// TIA Portal project "Boiler_DE_10_14GM" (V14)
// Паровой котел ДЕ-10-14ГМ

(* hardware
DEVICE "ET 200SP station_1"  ET 200SP-Station
   slot 0: "Rack_0"  Rack  6ES5 710-8MAx1
   slot 1: "PLC_1"  CPU 1510SP-1 PN  6ES7 510-1DJ01-0AB0  V2.1
   slot 2: "AI 8xI 2-,4-wire BA_1"  AI 8xI 2-,4-wire BA  6ES7 134-6GF00-0AA1  V1.0
      slot 1: "AI 8xI 2-,4-wire BA_1"  AI 8xI 2-,4-wire BA
   slot 3: "AI 8xI 2-,4-wire BA_2"  AI 8xI 2-,4-wire BA  6ES7 134-6GF00-0AA1  V1.0
      slot 1: "AI 8xI 2-,4-wire BA_2"  AI 8xI 2-,4-wire BA
   slot 4: "AI 8xI 2-,4-wire BA_3"  AI 8xI 2-,4-wire BA  6ES7 134-6GF00-0AA1  V1.0
      slot 1: "AI 8xI 2-,4-wire BA_3"  AI 8xI 2-,4-wire BA
   slot 5: "AI 8xI 2-,4-wire BA_4"  AI 8xI 2-,4-wire BA  6ES7 134-6GF00-0AA1  V1.0
      slot 1: "AI 8xI 2-,4-wire BA_4"  AI 8xI 2-,4-wire BA
   slot 6: "DI 16x24VDC ST_1"  DI 16x24VDC ST  6ES7 131-6BH00-0BA0  V1.1
      slot 1: "DI 16x24VDC ST_1"  DI 16x24VDC ST
   slot 7: "DI 16x24VDC ST_2"  DI 16x24VDC ST  6ES7 131-6BH00-0BA0  V1.1
      slot 1: "DI 16x24VDC ST_2"  DI 16x24VDC ST
   slot 8: "DI 16x24VDC ST_3"  DI 16x24VDC ST  6ES7 131-6BH00-0BA0  V1.1
      slot 1: "DI 16x24VDC ST_3"  DI 16x24VDC ST
   slot 9: "DI 16x24VDC ST_4"  DI 16x24VDC ST  6ES7 131-6BH00-0BA0  V1.1
      slot 1: "DI 16x24VDC ST_4"  DI 16x24VDC ST
   slot 10: "DI 16x24VDC ST_5"  DI 16x24VDC ST  6ES7 131-6BH00-0BA0  V1.1
      slot 1: "DI 16x24VDC ST_5"  DI 16x24VDC ST
   slot 11: "DI 16x24VDC ST_6"  DI 16x24VDC ST  6ES7 131-6BH00-0BA0  V1.1
      slot 1: "DI 16x24VDC ST_6"  DI 16x24VDC ST
   slot 12: "DQ 16x24VDC/0.5A ST_1"  DQ 16x24VDC/0.5A ST  6ES7 132-6BH00-0BA0  V1.1
      slot 1: "DQ 16x24VDC/0.5A ST_1"  DQ 16x24VDC/0.5A ST
   slot 13: "DQ 16x24VDC/0.5A ST_2"  DQ 16x24VDC/0.5A ST  6ES7 132-6BH00-0BA0  V1.1
      slot 1: "DQ 16x24VDC/0.5A ST_2"  DQ 16x24VDC/0.5A ST
   slot 14: "DQ 16x24VDC/0.5A ST_3"  DQ 16x24VDC/0.5A ST  6ES7 132-6BH00-0BA0  V1.1
      slot 1: "DQ 16x24VDC/0.5A ST_3"  DQ 16x24VDC/0.5A ST
   slot 15: "AQ 4xU/I ST_1"  AQ 4xU/I ST  6ES7 135-6HD00-0BA1  V1.1
      slot 1: "AQ 4xU/I ST_1"  AQ 4xU/I ST
   slot 16: "Server module_1"  Server module  6ES7 193-6PA00-0AA0  V1.1
      slot 1: "Server module_1"  Server module
   slot 127: "BA 2xRJ45"  BA 2xRJ45  6ES7 193-6AR00-0AA0  V0.0
      slot 32769: "Port_1"  6ES7 193-6AR00-0AA0
      slot 32770: "Port_2"  6ES7 193-6AR00-0AA0
*)

// ===== PLC "PLC_1"  CPU 1510SP-1 PN =====

VAR_GLOBAL   // PLC tag table "Default tag table"
   "Module01Chanel1_DI" AT %I0.0 : Bool;
   "Module01Chanel2_DI" AT %I0.1 : Bool;
   "Module01Chanel3_DI" AT %I0.2 : Bool;
   "Module01Chanel4_DI" AT %I0.3 : Bool;
   "Module01Chanel5_DI" AT %I0.4 : Bool;
   "Module01Chanel6_DI" AT %I0.5 : Bool;
   "Module01Chanel7_DI" AT %I0.6 : Bool;
   "Module01Chanel8_DI" AT %I0.7 : Bool;
   "Module01Chanel9_DI" AT %I1.0 : Bool;
   "Module01Chanel10_DI" AT %I1.1 : Bool;
   "Module01Chanel11_DI" AT %I1.2 : Bool;
   "Module01Chanel12_DI" AT %I1.3 : Bool;
   "Module01Chanel13_DI" AT %I1.4 : Bool;
   "Module01Chanel14_DI" AT %I1.5 : Bool;
   "Module01Chanel15_DI" AT %I1.6 : Bool;
   "Module01Chanel16_DI" AT %I1.7 : Bool;
   "Module01Chanel1_DO" AT %Q0.0 : Bool;
   "Module01Chanel2_DO" AT %Q0.1 : Bool;
   "Module01Chanel3_DO" AT %Q0.2 : Bool;
   "Module01Chanel4_DO" AT %Q0.3 : Bool;
   "Module01Chanel5_DO" AT %Q0.4 : Bool;
   "Module01Chanel6_DO" AT %Q0.5 : Bool;
   "Module01Chanel7_DO" AT %Q0.6 : Bool;
   "Module01Chanel8_DO" AT %Q0.7 : Bool;
   "Module01Chanel9_DO" AT %Q1.0 : Bool;
   "Module01Chanel10_DO" AT %Q1.1 : Bool;
   "Module01Chanel11_DO" AT %Q1.2 : Bool;
   "Module01Chanel12_DO" AT %Q1.3 : Bool;
   "Module01Chanel13_DO" AT %Q1.4 : Bool;
   "Module01Chanel14_DO" AT %Q1.5 : Bool;
   "Module01Chanel15_DO" AT %Q1.6 : Bool;
   "Module01Chanel16_DO" AT %Q1.7 : Bool;
   "Module01Chanel1_AI" AT %IW0 : Int;
   "Module01Chanel2_AI" AT %IW2 : Int;
   "Module01Chanel3_AI" AT %IW4 : Int;
   "Module01Chanel4_AI" AT %IW6 : Int;
   "Module01Chanel5_AI" AT %IW8 : Int;
   "Module01Chanel6_AI" AT %IW10 : Int;
   "Module01Chanel7_AI" AT %IW12 : Int;
   "Module01Chanel8_AI" AT %IW14 : Int;
   "Module01Chanel1_AO" AT %QW0 : Int;
   "Module01Chanel2_AO" AT %QW2 : Int;
   "Module01Chanel3_AO" AT %QW4 : Int;
   "Module01Chanel4_AO" AT %QW6 : Int;
   "Module02Chanel1_DI" AT %I16.0 : Bool;
   "Module02Chanel2_DI" AT %I16.1 : Bool;
   "Module02Chanel3_DI" AT %I16.2 : Bool;
   "Module02Chanel4_DI" AT %I16.3 : Bool;
   "Module02Chanel5_DI" AT %I16.4 : Bool;
   "Module02Chanel6_DI" AT %I16.5 : Bool;
   "Module02Chanel7_DI" AT %I16.6 : Bool;
   "Module02Chanel8_DI" AT %I16.7 : Bool;
   "Module02Chanel9_DI" AT %I17.0 : Bool;
   "Module02Chanel10_DI" AT %I17.1 : Bool;
   "Module02Chanel11_DI" AT %I17.2 : Bool;
   "Module02Chanel12_DI" AT %I17.3 : Bool;
   "Module02Chanel13_DI" AT %I17.4 : Bool;
   "Module02Chanel14_DI" AT %I17.5 : Bool;
   "Module02Chanel15_DI" AT %I17.6 : Bool;
   "Module02Chanel16_DI" AT %I17.7 : Bool;
   "Module02Chanel1_DO" AT %Q16.0 : Bool;
   "Module02Chanel2_DO" AT %Q16.1 : Bool;
   "Module02Chanel3_DO" AT %Q16.2 : Bool;
   "Module02Chanel4_DO" AT %Q16.3 : Bool;
   "Module02Chanel5_DO" AT %Q16.4 : Bool;
   "Module02Chanel6_DO" AT %Q16.5 : Bool;
   "Module02Chanel7_DO" AT %Q16.6 : Bool;
   "Module02Chanel8_DO" AT %Q16.7 : Bool;
   "Module02Chanel9_DO" AT %Q17.0 : Bool;
   "Module02Chanel10_DO" AT %Q17.1 : Bool;
   "Module02Chanel11_DO" AT %Q17.2 : Bool;
   "Module02Chanel12_DO" AT %Q17.3 : Bool;
   "Module02Chanel13_DO" AT %Q17.4 : Bool;
   "Module02Chanel14_DO" AT %Q17.5 : Bool;
   "Module02Chanel15_DO" AT %Q17.6 : Bool;
   "Module02Chanel16_DO" AT %Q17.7 : Bool;
   "Module02Chanel1_AI" AT %IW16 : Int;
   "Module02Chanel2_AI" AT %IW18 : Int;
   "Module02Chanel3_AI" AT %IW20 : Int;
   "Module02Chanel4_AI" AT %IW22 : Int;
   "Module02Chanel5_AI" AT %IW24 : Int;
   "Module02Chanel6_AI" AT %IW26 : Int;
   "Module02Chanel7_AI" AT %IW28 : Int;
   "Module02Chanel8_AI" AT %IW30 : Int;
   "Module02Chanel1_AO" AT %QW16 : Int;
   "Module02Chanel2_AO" AT %QW18 : Int;
   "Module02Chanel3_AO" AT %QW20 : Int;
   "Module02Chanel4_AO" AT %QW22 : Int;
   "Module03Chanel1_DI" AT %I32.0 : Bool;
   "Module03Chanel2_DI" AT %I32.1 : Bool;
   "Module03Chanel3_DI" AT %I32.2 : Bool;
   "Module03Chanel4_DI" AT %I32.3 : Bool;
   "Module03Chanel5_DI" AT %I32.4 : Bool;
   "Module03Chanel6_DI" AT %I32.5 : Bool;
   "Module03Chanel7_DI" AT %I32.6 : Bool;
   "Module03Chanel8_DI" AT %I32.7 : Bool;
   "Module03Chanel9_DI" AT %I33.0 : Bool;
   "Module03Chanel10_DI" AT %I33.1 : Bool;
   "Module03Chanel11_DI" AT %I33.2 : Bool;
   "Module03Chanel12_DI" AT %I33.3 : Bool;
   "Module03Chanel13_DI" AT %I33.4 : Bool;
   "Module03Chanel14_DI" AT %I33.5 : Bool;
   "Module03Chanel15_DI" AT %I33.6 : Bool;
   "Module03Chanel16_DI" AT %I33.7 : Bool;
   "Module03Chanel1_DO" AT %Q32.0 : Bool;
   "Module03Chanel2_DO" AT %Q32.1 : Bool;
   "Module03Chanel3_DO" AT %Q32.2 : Bool;
   "Module03Chanel4_DO" AT %Q32.3 : Bool;
   "Module03Chanel5_DO" AT %Q32.4 : Bool;
   "Module03Chanel6_DO" AT %Q32.5 : Bool;
   "Module03Chanel7_DO" AT %Q32.6 : Bool;
   "Module03Chanel8_DO" AT %Q32.7 : Bool;
   "Module03Chanel9_DO" AT %Q33.0 : Bool;
   "Module03Chanel10_DO" AT %Q33.1 : Bool;
   "Module03Chanel11_DO" AT %Q33.2 : Bool;
   "Module03Chanel12_DO" AT %Q33.3 : Bool;
   "Module03Chanel13_DO" AT %Q33.4 : Bool;
   "Module03Chanel14_DO" AT %Q33.5 : Bool;
   "Module03Chanel15_DO" AT %Q33.6 : Bool;
   "Module03Chanel16_DO" AT %Q33.7 : Bool;
   "Module03Chanel1_AI" AT %IW32 : Int;
   "Module03Chanel2_AI" AT %IW34 : Int;
   "Module03Chanel3_AI" AT %IW36 : Int;
   "Module03Chanel4_AI" AT %IW38 : Int;
   "Module03Chanel5_AI" AT %IW40 : Int;
   "Module03Chanel6_AI" AT %IW42 : Int;
   "Module03Chanel7_AI" AT %IW44 : Int;
   "Module03Chanel8_AI" AT %IW46 : Int;
   "Module03Chanel1_AO" AT %QW32 : Int;
   "Module03Chanel2_AO" AT %QW34 : Int;
   "Module03Chanel3_AO" AT %QW36 : Int;
   "Module03Chanel4_AO" AT %QW38 : Int;
   "Module04Chanel1_DI" AT %I48.0 : Bool;
   "Module04Chanel2_DI" AT %I48.1 : Bool;
   "Module04Chanel3_DI" AT %I48.2 : Bool;
   "Module04Chanel4_DI" AT %I48.3 : Bool;
   "Module04Chanel5_DI" AT %I48.4 : Bool;
   "Module04Chanel6_DI" AT %I48.5 : Bool;
   "Module04Chanel7_DI" AT %I48.6 : Bool;
   "Module04Chanel8_DI" AT %I48.7 : Bool;
   "Module04Chanel9_DI" AT %I49.0 : Bool;
   "Module04Chanel10_DI" AT %I49.1 : Bool;
   "Module04Chanel11_DI" AT %I49.2 : Bool;
   "Module04Chanel12_DI" AT %I49.3 : Bool;
   "Module04Chanel13_DI" AT %I49.4 : Bool;
   "Module04Chanel14_DI" AT %I49.5 : Bool;
   "Module04Chanel15_DI" AT %I49.6 : Bool;
   "Module04Chanel16_DI" AT %I49.7 : Bool;
   "Module04Chanel1_DO" AT %Q48.0 : Bool;
   "Module04Chanel2_DO" AT %Q48.1 : Bool;
   "Module04Chanel3_DO" AT %Q48.2 : Bool;
   "Module04Chanel4_DO" AT %Q48.3 : Bool;
   "Module04Chanel5_DO" AT %Q48.4 : Bool;
   "Module04Chanel6_DO" AT %Q48.5 : Bool;
   "Module04Chanel7_DO" AT %Q48.6 : Bool;
   "Module04Chanel8_DO" AT %Q48.7 : Bool;
   "Module04Chanel9_DO" AT %Q49.0 : Bool;
   "Module04Chanel10_DO" AT %Q49.1 : Bool;
   "Module04Chanel11_DO" AT %Q49.2 : Bool;
   "Module04Chanel12_DO" AT %Q49.3 : Bool;
   "Module04Chanel13_DO" AT %Q49.4 : Bool;
   "Module04Chanel14_DO" AT %Q49.5 : Bool;
   "Module04Chanel15_DO" AT %Q49.6 : Bool;
   "Module04Chanel16_DO" AT %Q49.7 : Bool;
   "Module04Chanel1_AI" AT %IW48 : Int;
   "Module04Chanel2_AI" AT %IW50 : Int;
   "Module04Chanel3_AI" AT %IW52 : Int;
   "Module04Chanel4_AI" AT %IW54 : Int;
   "Module04Chanel5_AI" AT %IW56 : Int;
   "Module04Chanel6_AI" AT %IW58 : Int;
   "Module04Chanel7_AI" AT %IW60 : Int;
   "Module04Chanel8_AI" AT %IW62 : Int;
   "Module04Chanel1_AO" AT %QW48 : Int;
   "Module04Chanel2_AO" AT %QW50 : Int;
   "Module04Chanel3_AO" AT %QW52 : Int;
   "Module04Chanel4_AO" AT %QW54 : Int;
   "Module05Chanel1_DI" AT %I64.0 : Bool;
   "Module05Chanel2_DI" AT %I64.1 : Bool;
   "Module05Chanel3_DI" AT %I64.2 : Bool;
   "Module05Chanel4_DI" AT %I64.3 : Bool;
   "Module05Chanel5_DI" AT %I64.4 : Bool;
   "Module05Chanel6_DI" AT %I64.5 : Bool;
   "Module05Chanel7_DI" AT %I64.6 : Bool;
   "Module05Chanel8_DI" AT %I64.7 : Bool;
   "Module05Chanel9_DI" AT %I65.0 : Bool;
   "Module05Chanel10_DI" AT %I65.1 : Bool;
   "Module05Chanel11_DI" AT %I65.2 : Bool;
   "Module05Chanel12_DI" AT %I65.3 : Bool;
   "Module05Chanel13_DI" AT %I65.4 : Bool;
   "Module05Chanel14_DI" AT %I65.5 : Bool;
   "Module05Chanel15_DI" AT %I65.6 : Bool;
   "Module05Chanel16_DI" AT %I65.7 : Bool;
   "Module05Chanel1_DO" AT %Q64.0 : Bool;
   "Module05Chanel2_DO" AT %Q64.1 : Bool;
   "Module05Chanel3_DO" AT %Q64.2 : Bool;
   "Module05Chanel4_DO" AT %Q64.3 : Bool;
   "Module05Chanel5_DO" AT %Q64.4 : Bool;
   "Module05Chanel6_DO" AT %Q64.5 : Bool;
   "Module05Chanel7_DO" AT %Q64.6 : Bool;
   "Module05Chanel8_DO" AT %Q64.7 : Bool;
   "Module05Chanel9_DO" AT %Q65.0 : Bool;
   "Module05Chanel10_DO" AT %Q65.1 : Bool;
   "Module05Chanel11_DO" AT %Q65.2 : Bool;
   "Module05Chanel12_DO" AT %Q65.3 : Bool;
   "Module05Chanel13_DO" AT %Q65.4 : Bool;
   "Module05Chanel14_DO" AT %Q65.5 : Bool;
   "Module05Chanel15_DO" AT %Q65.6 : Bool;
   "Module05Chanel16_DO" AT %Q65.7 : Bool;
   "Module05Chanel1_AI" AT %IW64 : Int;
   "Module05Chanel2_AI" AT %IW66 : Int;
   "Module05Chanel3_AI" AT %IW68 : Int;
   "Module05Chanel4_AI" AT %IW70 : Int;
   "Module05Chanel5_AI" AT %IW72 : Int;
   "Module05Chanel6_AI" AT %IW74 : Int;
   "Module05Chanel7_AI" AT %IW76 : Int;
   "Module05Chanel8_AI" AT %IW78 : Int;
   "Module05Chanel1_AO" AT %QW64 : Int;
   "Module05Chanel2_AO" AT %QW66 : Int;
   "Module05Chanel3_AO" AT %QW68 : Int;
   "Module05Chanel4_AO" AT %QW70 : Int;
   "Module06Chanel1_DI" AT %I80.0 : Bool;
   "Module06Chanel2_DI" AT %I80.1 : Bool;
   "Module06Chanel3_DI" AT %I80.2 : Bool;
   "Module06Chanel4_DI" AT %I80.3 : Bool;
   "Module06Chanel5_DI" AT %I80.4 : Bool;
   "Module06Chanel6_DI" AT %I80.5 : Bool;
   "Module06Chanel7_DI" AT %I80.6 : Bool;
   "Module06Chanel8_DI" AT %I80.7 : Bool;
   "Module06Chanel9_DI" AT %I81.0 : Bool;
   "Module06Chanel10_DI" AT %I81.1 : Bool;
   "Module06Chanel11_DI" AT %I81.2 : Bool;
   "Module06Chanel12_DI" AT %I81.3 : Bool;
   "Module06Chanel13_DI" AT %I81.4 : Bool;
   "Module06Chanel14_DI" AT %I81.5 : Bool;
   "Module06Chanel15_DI" AT %I81.6 : Bool;
   "Module06Chanel16_DI" AT %I81.7 : Bool;
   "Module06Chanel1_DO" AT %Q80.0 : Bool;
   "Module06Chanel2_DO" AT %Q80.1 : Bool;
   "Module06Chanel3_DO" AT %Q80.2 : Bool;
   "Module06Chanel4_DO" AT %Q80.3 : Bool;
   "Module06Chanel5_DO" AT %Q80.4 : Bool;
   "Module06Chanel6_DO" AT %Q80.5 : Bool;
   "Module06Chanel7_DO" AT %Q80.6 : Bool;
   "Module06Chanel8_DO" AT %Q80.7 : Bool;
   "Module06Chanel9_DO" AT %Q81.0 : Bool;
   "Module06Chanel10_DO" AT %Q81.1 : Bool;
   "Module06Chanel11_DO" AT %Q81.2 : Bool;
   "Module06Chanel12_DO" AT %Q81.3 : Bool;
   "Module06Chanel13_DO" AT %Q81.4 : Bool;
   "Module06Chanel14_DO" AT %Q81.5 : Bool;
   "Module06Chanel15_DO" AT %Q81.6 : Bool;
   "Module06Chanel16_DO" AT %Q81.7 : Bool;
   "Module06Chanel1_AI" AT %IW80 : Int;
   "Module06Chanel2_AI" AT %IW82 : Int;
   "Module06Chanel3_AI" AT %IW84 : Int;
   "Module06Chanel4_AI" AT %IW86 : Int;
   "Module06Chanel5_AI" AT %IW88 : Int;
   "Module06Chanel6_AI" AT %IW90 : Int;
   "Module06Chanel7_AI" AT %IW92 : Int;
   "Module06Chanel8_AI" AT %IW94 : Int;
   "Module06Chanel1_AO" AT %QW80 : Int;
   "Module06Chanel2_AO" AT %QW82 : Int;
   "Module06Chanel3_AO" AT %QW84 : Int;
   "Module06Chanel4_AO" AT %QW86 : Int;
   "Module07Chanel1_DI" AT %I96.0 : Bool;
   "Module07Chanel2_DI" AT %I96.1 : Bool;
   "Module07Chanel3_DI" AT %I96.2 : Bool;
   "Module07Chanel4_DI" AT %I96.3 : Bool;
   "Module07Chanel5_DI" AT %I96.4 : Bool;
   "Module07Chanel6_DI" AT %I96.5 : Bool;
   "Module07Chanel7_DI" AT %I96.6 : Bool;
   "Module07Chanel8_DI" AT %I96.7 : Bool;
   "Module07Chanel9_DI" AT %I97.0 : Bool;
   "Module07Chanel10_DI" AT %I97.1 : Bool;
   "Module07Chanel11_DI" AT %I97.2 : Bool;
   "Module07Chanel12_DI" AT %I97.3 : Bool;
   "Module07Chanel13_DI" AT %I97.4 : Bool;
   "Module07Chanel14_DI" AT %I97.5 : Bool;
   "Module07Chanel15_DI" AT %I97.6 : Bool;
   "Module07Chanel16_DI" AT %I97.7 : Bool;
   "Module07Chanel1_DO" AT %Q96.0 : Bool;
   "Module07Chanel2_DO" AT %Q96.1 : Bool;
   "Module07Chanel3_DO" AT %Q96.2 : Bool;
   "Module07Chanel4_DO" AT %Q96.3 : Bool;
   "Module07Chanel5_DO" AT %Q96.4 : Bool;
   "Module07Chanel6_DO" AT %Q96.5 : Bool;
   "Module07Chanel7_DO" AT %Q96.6 : Bool;
   "Module07Chanel8_DO" AT %Q96.7 : Bool;
   "Module07Chanel9_DO" AT %Q97.0 : Bool;
   "Module07Chanel10_DO" AT %Q97.1 : Bool;
   "Module07Chanel11_DO" AT %Q97.2 : Bool;
   "Module07Chanel12_DO" AT %Q97.3 : Bool;
   "Module07Chanel13_DO" AT %Q97.4 : Bool;
   "Module07Chanel14_DO" AT %Q97.5 : Bool;
   "Module07Chanel15_DO" AT %Q97.6 : Bool;
   "Module07Chanel16_DO" AT %Q97.7 : Bool;
   "Module07Chanel1_AI" AT %IW96 : Int;
   "Module07Chanel2_AI" AT %IW98 : Int;
   "Module07Chanel3_AI" AT %IW100 : Int;
   "Module07Chanel4_AI" AT %IW102 : Int;
   "Module07Chanel5_AI" AT %IW104 : Int;
   "Module07Chanel6_AI" AT %IW106 : Int;
   "Module07Chanel7_AI" AT %IW108 : Int;
   "Module07Chanel8_AI" AT %IW110 : Int;
   "Module07Chanel1_AO" AT %QW96 : Int;
   "Module07Chanel2_AO" AT %QW98 : Int;
   "Module07Chanel3_AO" AT %QW100 : Int;
   "Module07Chanel4_AO" AT %QW102 : Int;
   "Module08Chanel1_DI" AT %I112.0 : Bool;
   "Module08Chanel2_DI" AT %I112.1 : Bool;
   "Module08Chanel3_DI" AT %I112.2 : Bool;
   "Module08Chanel4_DI" AT %I112.3 : Bool;
   "Module08Chanel5_DI" AT %I112.4 : Bool;
   "Module08Chanel6_DI" AT %I112.5 : Bool;
   "Module08Chanel7_DI" AT %I112.6 : Bool;
   "Module08Chanel8_DI" AT %I112.7 : Bool;
   "Module08Chanel9_DI" AT %I113.0 : Bool;
   "Module08Chanel10_DI" AT %I113.1 : Bool;
   "Module08Chanel11_DI" AT %I113.2 : Bool;
   "Module08Chanel12_DI" AT %I113.3 : Bool;
   "Module08Chanel13_DI" AT %I113.4 : Bool;
   "Module08Chanel14_DI" AT %I113.5 : Bool;
   "Module08Chanel15_DI" AT %I113.6 : Bool;
   "Module08Chanel16_DI" AT %I113.7 : Bool;
   "Module08Chanel1_DO" AT %Q112.0 : Bool;
   "Module08Chanel2_DO" AT %Q112.1 : Bool;
   "Module08Chanel3_DO" AT %Q112.2 : Bool;
   "Module08Chanel4_DO" AT %Q112.3 : Bool;
   "Module08Chanel5_DO" AT %Q112.4 : Bool;
   "Module08Chanel6_DO" AT %Q112.5 : Bool;
   "Module08Chanel7_DO" AT %Q112.6 : Bool;
   "Module08Chanel8_DO" AT %Q112.7 : Bool;
   "Module08Chanel9_DO" AT %Q113.0 : Bool;
   "Module08Chanel10_DO" AT %Q113.1 : Bool;
   "Module08Chanel11_DO" AT %Q113.2 : Bool;
   "Module08Chanel12_DO" AT %Q113.3 : Bool;
   "Module08Chanel13_DO" AT %Q113.4 : Bool;
   "Module08Chanel14_DO" AT %Q113.5 : Bool;
   "Module08Chanel15_DO" AT %Q113.6 : Bool;
   "Module08Chanel16_DO" AT %Q113.7 : Bool;
   "Module08Chanel1_AI" AT %IW112 : Int;
   "Module08Chanel2_AI" AT %IW114 : Int;
   "Module08Chanel3_AI" AT %IW116 : Int;
   "Module08Chanel4_AI" AT %IW118 : Int;
   "Module08Chanel5_AI" AT %IW120 : Int;
   "Module08Chanel6_AI" AT %IW122 : Int;
   "Module08Chanel7_AI" AT %IW124 : Int;
   "Module08Chanel8_AI" AT %IW126 : Int;
   "Module08Chanel1_AO" AT %QW112 : Int;
   "Module08Chanel2_AO" AT %QW114 : Int;
   "Module08Chanel3_AO" AT %QW116 : Int;
   "Module08Chanel4_AO" AT %QW118 : Int;
   "Module09Chanel1_DI" AT %I128.0 : Bool;
   "Module09Chanel2_DI" AT %I128.1 : Bool;
   "Module09Chanel3_DI" AT %I128.2 : Bool;
   "Module09Chanel4_DI" AT %I128.3 : Bool;
   "Module09Chanel5_DI" AT %I128.4 : Bool;
   "Module09Chanel6_DI" AT %I128.5 : Bool;
   "Module09Chanel7_DI" AT %I128.6 : Bool;
   "Module09Chanel8_DI" AT %I128.7 : Bool;
   "Module09Chanel9_DI" AT %I129.0 : Bool;
   "Module09Chanel10_DI" AT %I129.1 : Bool;
   "Module09Chanel11_DI" AT %I129.2 : Bool;
   "Module09Chanel12_DI" AT %I129.3 : Bool;
   "Module09Chanel13_DI" AT %I129.4 : Bool;
   "Module09Chanel14_DI" AT %I129.5 : Bool;
   "Module09Chanel15_DI" AT %I129.6 : Bool;
   "Module09Chanel16_DI" AT %I129.7 : Bool;
   "Module09Chanel1_DO" AT %Q128.0 : Bool;
   "Module09Chanel2_DO" AT %Q128.1 : Bool;
   "Module09Chanel3_DO" AT %Q128.2 : Bool;
   "Module09Chanel4_DO" AT %Q128.3 : Bool;
   "Module09Chanel5_DO" AT %Q128.4 : Bool;
   "Module09Chanel6_DO" AT %Q128.5 : Bool;
   "Module09Chanel7_DO" AT %Q128.6 : Bool;
   "Module09Chanel8_DO" AT %Q128.7 : Bool;
   "Module09Chanel9_DO" AT %Q129.0 : Bool;
   "Module09Chanel10_DO" AT %Q129.1 : Bool;
   "Module09Chanel11_DO" AT %Q129.2 : Bool;
   "Module09Chanel12_DO" AT %Q129.3 : Bool;
   "Module09Chanel13_DO" AT %Q129.4 : Bool;
   "Module09Chanel14_DO" AT %Q129.5 : Bool;
   "Module09Chanel15_DO" AT %Q129.6 : Bool;
   "Module09Chanel16_DO" AT %Q129.7 : Bool;
   "Module09Chanel1_AI" AT %IW128 : Int;
   "Module09Chanel2_AI" AT %IW130 : Int;
   "Module09Chanel3_AI" AT %IW132 : Int;
   "Module09Chanel4_AI" AT %IW134 : Int;
   "Module09Chanel5_AI" AT %IW136 : Int;
   "Module09Chanel6_AI" AT %IW138 : Int;
   "Module09Chanel7_AI" AT %IW140 : Int;
   "Module09Chanel8_AI" AT %IW142 : Int;
   "Module09Chanel1_AO" AT %QW128 : Int;
   "Module09Chanel2_AO" AT %QW130 : Int;
   "Module09Chanel3_AO" AT %QW132 : Int;
   "Module09Chanel4_AO" AT %QW134 : Int;
   "Module10Chanel1_DI" AT %I144.0 : Bool;
   "Module10Chanel2_DI" AT %I144.1 : Bool;
   "Module10Chanel3_DI" AT %I144.2 : Bool;
   "Module10Chanel4_DI" AT %I144.3 : Bool;
   "Module10Chanel5_DI" AT %I144.4 : Bool;
   "Module10Chanel6_DI" AT %I144.5 : Bool;
   "Module10Chanel7_DI" AT %I144.6 : Bool;
   "Module10Chanel8_DI" AT %I144.7 : Bool;
   "Module10Chanel9_DI" AT %I145.0 : Bool;
   "Module10Chanel10_DI" AT %I145.1 : Bool;
   "Module10Chanel11_DI" AT %I145.2 : Bool;
   "Module10Chanel12_DI" AT %I145.3 : Bool;
   "Module10Chanel13_DI" AT %I145.4 : Bool;
   "Module10Chanel14_DI" AT %I145.5 : Bool;
   "Module10Chanel15_DI" AT %I145.6 : Bool;
   "Module10Chanel16_DI" AT %I145.7 : Bool;
   "Module10Chanel1_DO" AT %Q144.0 : Bool;
   "Module10Chanel2_DO" AT %Q144.1 : Bool;
   "Module10Chanel3_DO" AT %Q144.2 : Bool;
   "Module10Chanel4_DO" AT %Q144.3 : Bool;
   "Module10Chanel5_DO" AT %Q144.4 : Bool;
   "Module10Chanel6_DO" AT %Q144.5 : Bool;
   "Module10Chanel7_DO" AT %Q144.6 : Bool;
   "Module10Chanel8_DO" AT %Q144.7 : Bool;
   "Module10Chanel9_DO" AT %Q145.0 : Bool;
   "Module10Chanel10_DO" AT %Q145.1 : Bool;
   "Module10Chanel11_DO" AT %Q145.2 : Bool;
   "Module10Chanel12_DO" AT %Q145.3 : Bool;
   "Module10Chanel13_DO" AT %Q145.4 : Bool;
   "Module10Chanel14_DO" AT %Q145.5 : Bool;
   "Module10Chanel15_DO" AT %Q145.6 : Bool;
   "Module10Chanel16_DO" AT %Q145.7 : Bool;
   "Module10Chanel1_AI" AT %IW144 : Int;
   "Module10Chanel2_AI" AT %IW146 : Int;
   "Module10Chanel3_AI" AT %IW148 : Int;
   "Module10Chanel4_AI" AT %IW150 : Int;
   "Module10Chanel5_AI" AT %IW152 : Int;
   "Module10Chanel6_AI" AT %IW154 : Int;
   "Module10Chanel7_AI" AT %IW156 : Int;
   "Module10Chanel8_AI" AT %IW158 : Int;
   "Module10Chanel1_AO" AT %QW144 : Int;
   "Module10Chanel2_AO" AT %QW146 : Int;
   "Module10Chanel3_AO" AT %QW148 : Int;
   "Module10Chanel4_AO" AT %QW150 : Int;
   "Module11Chanel1_DI" AT %I160.0 : Bool;
   "Module11Chanel2_DI" AT %I160.1 : Bool;
   "Module11Chanel3_DI" AT %I160.2 : Bool;
   "Module11Chanel4_DI" AT %I160.3 : Bool;
   "Module11Chanel5_DI" AT %I160.4 : Bool;
   "Module11Chanel6_DI" AT %I160.5 : Bool;
   "Module11Chanel7_DI" AT %I160.6 : Bool;
   "Module11Chanel8_DI" AT %I160.7 : Bool;
   "Module11Chanel9_DI" AT %I161.0 : Bool;
   "Module11Chanel10_DI" AT %I161.1 : Bool;
   "Module11Chanel11_DI" AT %I161.2 : Bool;
   "Module11Chanel12_DI" AT %I161.3 : Bool;
   "Module11Chanel13_DI" AT %I161.4 : Bool;
   "Module11Chanel14_DI" AT %I161.5 : Bool;
   "Module11Chanel15_DI" AT %I161.6 : Bool;
   "Module11Chanel16_DI" AT %I161.7 : Bool;
   "Module11Chanel1_DO" AT %Q160.0 : Bool;
   "Module11Chanel2_DO" AT %Q160.1 : Bool;
   "Module11Chanel3_DO" AT %Q160.2 : Bool;
   "Module11Chanel4_DO" AT %Q160.3 : Bool;
   "Module11Chanel5_DO" AT %Q160.4 : Bool;
   "Module11Chanel6_DO" AT %Q160.5 : Bool;
   "Module11Chanel7_DO" AT %Q160.6 : Bool;
   "Module11Chanel8_DO" AT %Q160.7 : Bool;
   "Module11Chanel9_DO" AT %Q161.0 : Bool;
   "Module11Chanel10_DO" AT %Q161.1 : Bool;
   "Module11Chanel11_DO" AT %Q161.2 : Bool;
   "Module11Chanel12_DO" AT %Q161.3 : Bool;
   "Module11Chanel13_DO" AT %Q161.4 : Bool;
   "Module11Chanel14_DO" AT %Q161.5 : Bool;
   "Module11Chanel15_DO" AT %Q161.6 : Bool;
   "Module11Chanel16_DO" AT %Q161.7 : Bool;
   "Module11Chanel1_AI" AT %IW160 : Int;
   "Module11Chanel2_AI" AT %IW162 : Int;
   "Module11Chanel3_AI" AT %IW164 : Int;
   "Module11Chanel4_AI" AT %IW166 : Int;
   "Module11Chanel5_AI" AT %IW168 : Int;
   "Module11Chanel6_AI" AT %IW170 : Int;
   "Module11Chanel7_AI" AT %IW172 : Int;
   "Module11Chanel8_AI" AT %IW174 : Int;
   "Module11Chanel1_AO" AT %QW160 : Int;
   "Module11Chanel2_AO" AT %QW162 : Int;
   "Module11Chanel3_AO" AT %QW164 : Int;
   "Module11Chanel4_AO" AT %QW166 : Int;
   "Module12Chanel1_DI" AT %I176.0 : Bool;
   "Module12Chanel2_DI" AT %I176.1 : Bool;
   "Module12Chanel3_DI" AT %I176.2 : Bool;
   "Module12Chanel4_DI" AT %I176.3 : Bool;
   "Module12Chanel5_DI" AT %I176.4 : Bool;
   "Module12Chanel6_DI" AT %I176.5 : Bool;
   "Module12Chanel7_DI" AT %I176.6 : Bool;
   "Module12Chanel8_DI" AT %I176.7 : Bool;
   "Module12Chanel9_DI" AT %I177.0 : Bool;
   "Module12Chanel10_DI" AT %I177.1 : Bool;
   "Module12Chanel11_DI" AT %I177.2 : Bool;
   "Module12Chanel12_DI" AT %I177.3 : Bool;
   "Module12Chanel13_DI" AT %I177.4 : Bool;
   "Module12Chanel14_DI" AT %I177.5 : Bool;
   "Module12Chanel15_DI" AT %I177.6 : Bool;
   "Module12Chanel16_DI" AT %I177.7 : Bool;
   "Module12Chanel1_DO" AT %Q176.0 : Bool;
   "Module12Chanel2_DO" AT %Q176.1 : Bool;
   "Module12Chanel3_DO" AT %Q176.2 : Bool;
   "Module12Chanel4_DO" AT %Q176.3 : Bool;
   "Module12Chanel5_DO" AT %Q176.4 : Bool;
   "Module12Chanel6_DO" AT %Q176.5 : Bool;
   "Module12Chanel7_DO" AT %Q176.6 : Bool;
   "Module12Chanel8_DO" AT %Q176.7 : Bool;
   "Module12Chanel9_DO" AT %Q177.0 : Bool;
   "Module12Chanel10_DO" AT %Q177.1 : Bool;
   "Module12Chanel11_DO" AT %Q177.2 : Bool;
   "Module12Chanel12_DO" AT %Q177.3 : Bool;
   "Module12Chanel13_DO" AT %Q177.4 : Bool;
   "Module12Chanel14_DO" AT %Q177.5 : Bool;
   "Module12Chanel15_DO" AT %Q177.6 : Bool;
   "Module12Chanel16_DO" AT %Q177.7 : Bool;
   "Module12Chanel1_AI" AT %IW176 : Int;
   "Module12Chanel2_AI" AT %IW178 : Int;
   "Module12Chanel3_AI" AT %IW180 : Int;
   "Module12Chanel4_AI" AT %IW182 : Int;
   "Module12Chanel5_AI" AT %IW184 : Int;
   "Module12Chanel6_AI" AT %IW186 : Int;
   "Module12Chanel7_AI" AT %IW188 : Int;
   "Module12Chanel8_AI" AT %IW190 : Int;
   "Module12Chanel1_AO" AT %QW176 : Int;
   "Module12Chanel2_AO" AT %QW178 : Int;
   "Module12Chanel3_AO" AT %QW180 : Int;
   "Module12Chanel4_AO" AT %QW182 : Int;
   "Module13Chanel1_DI" AT %I192.0 : Bool;
   "Module13Chanel2_DI" AT %I192.1 : Bool;
   "Module13Chanel3_DI" AT %I192.2 : Bool;
   "Module13Chanel4_DI" AT %I192.3 : Bool;
   "Module13Chanel5_DI" AT %I192.4 : Bool;
   "Module13Chanel6_DI" AT %I192.5 : Bool;
   "Module13Chanel7_DI" AT %I192.6 : Bool;
   "Module13Chanel8_DI" AT %I192.7 : Bool;
   "Module13Chanel9_DI" AT %I193.0 : Bool;
   "Module13Chanel10_DI" AT %I193.1 : Bool;
   "Module13Chanel11_DI" AT %I193.2 : Bool;
   "Module13Chanel12_DI" AT %I193.3 : Bool;
   "Module13Chanel13_DI" AT %I193.4 : Bool;
   "Module13Chanel14_DI" AT %I193.5 : Bool;
   "Module13Chanel15_DI" AT %I193.6 : Bool;
   "Module13Chanel16_DI" AT %I193.7 : Bool;
   "Module13Chanel1_DO" AT %Q192.0 : Bool;
   "Module13Chanel2_DO" AT %Q192.1 : Bool;
   "Module13Chanel3_DO" AT %Q192.2 : Bool;
   "Module13Chanel4_DO" AT %Q192.3 : Bool;
   "Module13Chanel5_DO" AT %Q192.4 : Bool;
   "Module13Chanel6_DO" AT %Q192.5 : Bool;
   "Module13Chanel7_DO" AT %Q192.6 : Bool;
   "Module13Chanel8_DO" AT %Q192.7 : Bool;
   "Module13Chanel9_DO" AT %Q193.0 : Bool;
   "Module13Chanel10_DO" AT %Q193.1 : Bool;
   "Module13Chanel11_DO" AT %Q193.2 : Bool;
   "Module13Chanel12_DO" AT %Q193.3 : Bool;
   "Module13Chanel13_DO" AT %Q193.4 : Bool;
   "Module13Chanel14_DO" AT %Q193.5 : Bool;
   "Module13Chanel15_DO" AT %Q193.6 : Bool;
   "Module13Chanel16_DO" AT %Q193.7 : Bool;
   "Module13Chanel1_AI" AT %IW192 : Int;
   "Module13Chanel2_AI" AT %IW194 : Int;
   "Module13Chanel3_AI" AT %IW196 : Int;
   "Module13Chanel4_AI" AT %IW198 : Int;
   "Module13Chanel5_AI" AT %IW200 : Int;
   "Module13Chanel6_AI" AT %IW202 : Int;
   "Module13Chanel7_AI" AT %IW204 : Int;
   "Module13Chanel8_AI" AT %IW206 : Int;
   "Module13Chanel1_AO" AT %QW192 : Int;
   "Module13Chanel2_AO" AT %QW194 : Int;
   "Module13Chanel3_AO" AT %QW196 : Int;
   "Module13Chanel4_AO" AT %QW198 : Int;
   "Module14Chanel1_DI" AT %I208.0 : Bool;
   "Module14Chanel2_DI" AT %I208.1 : Bool;
   "Module14Chanel3_DI" AT %I208.2 : Bool;
   "Module14Chanel4_DI" AT %I208.3 : Bool;
   "Module14Chanel5_DI" AT %I208.4 : Bool;
   "Module14Chanel6_DI" AT %I208.5 : Bool;
   "Module14Chanel7_DI" AT %I208.6 : Bool;
   "Module14Chanel8_DI" AT %I208.7 : Bool;
   "Module14Chanel9_DI" AT %I209.0 : Bool;
   "Module14Chanel10_DI" AT %I209.1 : Bool;
   "Module14Chanel11_DI" AT %I209.2 : Bool;
   "Module14Chanel12_DI" AT %I209.3 : Bool;
   "Module14Chanel13_DI" AT %I209.4 : Bool;
   "Module14Chanel14_DI" AT %I209.5 : Bool;
   "Module14Chanel15_DI" AT %I209.6 : Bool;
   "Module14Chanel16_DI" AT %I209.7 : Bool;
   "Module14Chanel1_DO" AT %Q208.0 : Bool;
   "Module14Chanel2_DO" AT %Q208.1 : Bool;
   "Module14Chanel3_DO" AT %Q208.2 : Bool;
   "Module14Chanel4_DO" AT %Q208.3 : Bool;
   "Module14Chanel5_DO" AT %Q208.4 : Bool;
   "Module14Chanel6_DO" AT %Q208.5 : Bool;
   "Module14Chanel7_DO" AT %Q208.6 : Bool;
   "Module14Chanel8_DO" AT %Q208.7 : Bool;
   "Module14Chanel9_DO" AT %Q209.0 : Bool;
   "Module14Chanel10_DO" AT %Q209.1 : Bool;
   "Module14Chanel11_DO" AT %Q209.2 : Bool;
   "Module14Chanel12_DO" AT %Q209.3 : Bool;
   "Module14Chanel13_DO" AT %Q209.4 : Bool;
   "Module14Chanel14_DO" AT %Q209.5 : Bool;
   "Module14Chanel15_DO" AT %Q209.6 : Bool;
   "Module14Chanel16_DO" AT %Q209.7 : Bool;
   "Module14Chanel1_AI" AT %IW208 : Int;
   "Module14Chanel2_AI" AT %IW210 : Int;
   "Module14Chanel3_AI" AT %IW212 : Int;
   "Module14Chanel4_AI" AT %IW214 : Int;
   "Module14Chanel5_AI" AT %IW216 : Int;
   "Module14Chanel6_AI" AT %IW218 : Int;
   "Module14Chanel7_AI" AT %IW220 : Int;
   "Module14Chanel8_AI" AT %IW222 : Int;
   "Module14Chanel1_AO" AT %QW208 : Int;
   "Module14Chanel2_AO" AT %QW210 : Int;
   "Module14Chanel3_AO" AT %QW212 : Int;
   "Module14Chanel4_AO" AT %QW214 : Int;
   "Module15Chanel1_DI" AT %I224.0 : Bool;
   "Module15Chanel2_DI" AT %I224.1 : Bool;
   "Module15Chanel3_DI" AT %I224.2 : Bool;
   "Module15Chanel4_DI" AT %I224.3 : Bool;
   "Module15Chanel5_DI" AT %I224.4 : Bool;
   "Module15Chanel6_DI" AT %I224.5 : Bool;
   "Module15Chanel7_DI" AT %I224.6 : Bool;
   "Module15Chanel8_DI" AT %I224.7 : Bool;
   "Module15Chanel9_DI" AT %I225.0 : Bool;
   "Module15Chanel10_DI" AT %I225.1 : Bool;
   "Module15Chanel11_DI" AT %I225.2 : Bool;
   "Module15Chanel12_DI" AT %I225.3 : Bool;
   "Module15Chanel13_DI" AT %I225.4 : Bool;
   "Module15Chanel14_DI" AT %I225.5 : Bool;
   "Module15Chanel15_DI" AT %I225.6 : Bool;
   "Module15Chanel16_DI" AT %I225.7 : Bool;
   "Module15Chanel1_DO" AT %Q224.0 : Bool;
   "Module15Chanel2_DO" AT %Q224.1 : Bool;
   "Module15Chanel3_DO" AT %Q224.2 : Bool;
   "Module15Chanel4_DO" AT %Q224.3 : Bool;
   "Module15Chanel5_DO" AT %Q224.4 : Bool;
   "Module15Chanel6_DO" AT %Q224.5 : Bool;
   "Module15Chanel7_DO" AT %Q224.6 : Bool;
   "Module15Chanel8_DO" AT %Q224.7 : Bool;
   "Module15Chanel9_DO" AT %Q225.0 : Bool;
   "Module15Chanel10_DO" AT %Q225.1 : Bool;
   "Module15Chanel11_DO" AT %Q225.2 : Bool;
   "Module15Chanel12_DO" AT %Q225.3 : Bool;
   "Module15Chanel13_DO" AT %Q225.4 : Bool;
   "Module15Chanel14_DO" AT %Q225.5 : Bool;
   "Module15Chanel15_DO" AT %Q225.6 : Bool;
   "Module15Chanel16_DO" AT %Q225.7 : Bool;
   "Module15Chanel1_AI" AT %IW224 : Int;
   "Module15Chanel2_AI" AT %IW226 : Int;
   "Module15Chanel3_AI" AT %IW228 : Int;
   "Module15Chanel4_AI" AT %IW230 : Int;
   "Module15Chanel5_AI" AT %IW232 : Int;
   "Module15Chanel6_AI" AT %IW234 : Int;
   "Module15Chanel7_AI" AT %IW236 : Int;
   "Module15Chanel8_AI" AT %IW238 : Int;
   "Module15Chanel1_AO" AT %QW224 : Int;
   "Module15Chanel2_AO" AT %QW226 : Int;
   "Module15Chanel3_AO" AT %QW228 : Int;
   "Module15Chanel4_AO" AT %QW230 : Int;
   "Module16Chanel1_DI" AT %I240.0 : Bool;
   "Module16Chanel2_DI" AT %I240.1 : Bool;
   "Module16Chanel3_DI" AT %I240.2 : Bool;
   "Module16Chanel4_DI" AT %I240.3 : Bool;
   "Module16Chanel5_DI" AT %I240.4 : Bool;
   "Module16Chanel6_DI" AT %I240.5 : Bool;
   "Module16Chanel7_DI" AT %I240.6 : Bool;
   "Module16Chanel8_DI" AT %I240.7 : Bool;
   "Module16Chanel9_DI" AT %I241.0 : Bool;
   "Module16Chanel10_DI" AT %I241.1 : Bool;
   "Module16Chanel11_DI" AT %I241.2 : Bool;
   "Module16Chanel12_DI" AT %I241.3 : Bool;
   "Module16Chanel13_DI" AT %I241.4 : Bool;
   "Module16Chanel14_DI" AT %I241.5 : Bool;
   "Module16Chanel15_DI" AT %I241.6 : Bool;
   "Module16Chanel16_DI" AT %I241.7 : Bool;
   "Module16Chanel1_DO" AT %Q240.0 : Bool;
   "Module16Chanel2_DO" AT %Q240.1 : Bool;
   "Module16Chanel3_DO" AT %Q240.2 : Bool;
   "Module16Chanel4_DO" AT %Q240.3 : Bool;
   "Module16Chanel5_DO" AT %Q240.4 : Bool;
   "Module16Chanel6_DO" AT %Q240.5 : Bool;
   "Module16Chanel7_DO" AT %Q240.6 : Bool;
   "Module16Chanel8_DO" AT %Q240.7 : Bool;
   "Module16Chanel9_DO" AT %Q241.0 : Bool;
   "Module16Chanel10_DO" AT %Q241.1 : Bool;
   "Module16Chanel11_DO" AT %Q241.2 : Bool;
   "Module16Chanel12_DO" AT %Q241.3 : Bool;
   "Module16Chanel13_DO" AT %Q241.4 : Bool;
   "Module16Chanel14_DO" AT %Q241.5 : Bool;
   "Module16Chanel15_DO" AT %Q241.6 : Bool;
   "Module16Chanel16_DO" AT %Q241.7 : Bool;
   "Module16Chanel1_AI" AT %IW240 : Int;
   "Module16Chanel2_AI" AT %IW242 : Int;
   "Module16Chanel3_AI" AT %IW244 : Int;
   "Module16Chanel4_AI" AT %IW246 : Int;
   "Module16Chanel5_AI" AT %IW248 : Int;
   "Module16Chanel6_AI" AT %IW250 : Int;
   "Module16Chanel7_AI" AT %IW252 : Int;
   "Module16Chanel8_AI" AT %IW254 : Int;
   "Module16Chanel1_AO" AT %QW240 : Int;
   "Module16Chanel2_AO" AT %QW242 : Int;
   "Module16Chanel3_AO" AT %QW244 : Int;
   "Module16Chanel4_AO" AT %QW246 : Int;
   "Module17Chanel1_DI" AT %I256.0 : Bool;
   "Module17Chanel2_DI" AT %I256.1 : Bool;
   "Module17Chanel3_DI" AT %I256.2 : Bool;
   "Module17Chanel4_DI" AT %I256.3 : Bool;
   "Module17Chanel5_DI" AT %I256.4 : Bool;
   "Module17Chanel6_DI" AT %I256.5 : Bool;
   "Module17Chanel7_DI" AT %I256.6 : Bool;
   "Module17Chanel8_DI" AT %I256.7 : Bool;
   "Module17Chanel9_DI" AT %I257.0 : Bool;
   "Module17Chanel10_DI" AT %I257.1 : Bool;
   "Module17Chanel11_DI" AT %I257.2 : Bool;
   "Module17Chanel12_DI" AT %I257.3 : Bool;
   "Module17Chanel13_DI" AT %I257.4 : Bool;
   "Module17Chanel14_DI" AT %I257.5 : Bool;
   "Module17Chanel15_DI" AT %I257.6 : Bool;
   "Module17Chanel16_DI" AT %I257.7 : Bool;
   "Module17Chanel1_DO" AT %Q256.0 : Bool;
   "Module17Chanel2_DO" AT %Q256.1 : Bool;
   "Module17Chanel3_DO" AT %Q256.2 : Bool;
   "Module17Chanel4_DO" AT %Q256.3 : Bool;
   "Module17Chanel5_DO" AT %Q256.4 : Bool;
   "Module17Chanel6_DO" AT %Q256.5 : Bool;
   "Module17Chanel7_DO" AT %Q256.6 : Bool;
   "Module17Chanel8_DO" AT %Q256.7 : Bool;
   "Module17Chanel9_DO" AT %Q257.0 : Bool;
   "Module17Chanel10_DO" AT %Q257.1 : Bool;
   "Module17Chanel11_DO" AT %Q257.2 : Bool;
   "Module17Chanel12_DO" AT %Q257.3 : Bool;
   "Module17Chanel13_DO" AT %Q257.4 : Bool;
   "Module17Chanel14_DO" AT %Q257.5 : Bool;
   "Module17Chanel15_DO" AT %Q257.6 : Bool;
   "Module17Chanel16_DO" AT %Q257.7 : Bool;
   "Module17Chanel1_AI" AT %IW256 : Int;
   "Module17Chanel2_AI" AT %IW258 : Int;
   "Module17Chanel3_AI" AT %IW260 : Int;
   "Module17Chanel4_AI" AT %IW262 : Int;
   "Module17Chanel5_AI" AT %IW264 : Int;
   "Module17Chanel6_AI" AT %IW266 : Int;
   "Module17Chanel7_AI" AT %IW268 : Int;
   "Module17Chanel8_AI" AT %IW270 : Int;
   "Module17Chanel1_AO" AT %QW256 : Int;
   "Module17Chanel2_AO" AT %QW258 : Int;
   "Module17Chanel3_AO" AT %QW260 : Int;
   "Module17Chanel4_AO" AT %QW262 : Int;
   "Module18Chanel1_DI" AT %I272.0 : Bool;
   "Module18Chanel2_DI" AT %I272.1 : Bool;
   "Module18Chanel3_DI" AT %I272.2 : Bool;
   "Module18Chanel4_DI" AT %I272.3 : Bool;
   "Module18Chanel5_DI" AT %I272.4 : Bool;
   "Module18Chanel6_DI" AT %I272.5 : Bool;
   "Module18Chanel7_DI" AT %I272.6 : Bool;
   "Module18Chanel8_DI" AT %I272.7 : Bool;
   "Module18Chanel9_DI" AT %I273.0 : Bool;
   "Module18Chanel10_DI" AT %I273.1 : Bool;
   "Module18Chanel11_DI" AT %I273.2 : Bool;
   "Module18Chanel12_DI" AT %I273.3 : Bool;
   "Module18Chanel13_DI" AT %I273.4 : Bool;
   "Module18Chanel14_DI" AT %I273.5 : Bool;
   "Module18Chanel15_DI" AT %I273.6 : Bool;
   "Module18Chanel16_DI" AT %I273.7 : Bool;
   "Module18Chanel1_DO" AT %Q272.0 : Bool;
   "Module18Chanel2_DO" AT %Q272.1 : Bool;
   "Module18Chanel3_DO" AT %Q272.2 : Bool;
   "Module18Chanel4_DO" AT %Q272.3 : Bool;
   "Module18Chanel5_DO" AT %Q272.4 : Bool;
   "Module18Chanel6_DO" AT %Q272.5 : Bool;
   "Module18Chanel7_DO" AT %Q272.6 : Bool;
   "Module18Chanel8_DO" AT %Q272.7 : Bool;
   "Module18Chanel9_DO" AT %Q273.0 : Bool;
   "Module18Chanel10_DO" AT %Q273.1 : Bool;
   "Module18Chanel11_DO" AT %Q273.2 : Bool;
   "Module18Chanel12_DO" AT %Q273.3 : Bool;
   "Module18Chanel13_DO" AT %Q273.4 : Bool;
   "Module18Chanel14_DO" AT %Q273.5 : Bool;
   "Module18Chanel15_DO" AT %Q273.6 : Bool;
   "Module18Chanel16_DO" AT %Q273.7 : Bool;
   "Module18Chanel1_AI" AT %IW272 : Int;
   "Module18Chanel2_AI" AT %IW274 : Int;
   "Module18Chanel3_AI" AT %IW276 : Int;
   "Module18Chanel4_AI" AT %IW278 : Int;
   "Module18Chanel5_AI" AT %IW280 : Int;
   "Module18Chanel6_AI" AT %IW282 : Int;
   "Module18Chanel7_AI" AT %IW284 : Int;
   "Module18Chanel8_AI" AT %IW286 : Int;
   "Module18Chanel1_AO" AT %QW272 : Int;
   "Module18Chanel2_AO" AT %QW274 : Int;
   "Module18Chanel3_AO" AT %QW276 : Int;
   "Module18Chanel4_AO" AT %QW278 : Int;
   "Module19Chanel1_DI" AT %I288.0 : Bool;
   "Module19Chanel2_DI" AT %I288.1 : Bool;
   "Module19Chanel3_DI" AT %I288.2 : Bool;
   "Module19Chanel4_DI" AT %I288.3 : Bool;
   "Module19Chanel5_DI" AT %I288.4 : Bool;
   "Module19Chanel6_DI" AT %I288.5 : Bool;
   "Module19Chanel7_DI" AT %I288.6 : Bool;
   "Module19Chanel8_DI" AT %I288.7 : Bool;
   "Module19Chanel9_DI" AT %I289.0 : Bool;
   "Module19Chanel10_DI" AT %I289.1 : Bool;
   "Module19Chanel11_DI" AT %I289.2 : Bool;
   "Module19Chanel12_DI" AT %I289.3 : Bool;
   "Module19Chanel13_DI" AT %I289.4 : Bool;
   "Module19Chanel14_DI" AT %I289.5 : Bool;
   "Module19Chanel15_DI" AT %I289.6 : Bool;
   "Module19Chanel16_DI" AT %I289.7 : Bool;
   "Module19Chanel1_DO" AT %Q288.0 : Bool;
   "Module19Chanel2_DO" AT %Q288.1 : Bool;
   "Module19Chanel3_DO" AT %Q288.2 : Bool;
   "Module19Chanel4_DO" AT %Q288.3 : Bool;
   "Module19Chanel5_DO" AT %Q288.4 : Bool;
   "Module19Chanel6_DO" AT %Q288.5 : Bool;
   "Module19Chanel7_DO" AT %Q288.6 : Bool;
   "Module19Chanel8_DO" AT %Q288.7 : Bool;
   "Module19Chanel9_DO" AT %Q289.0 : Bool;
   "Module19Chanel10_DO" AT %Q289.1 : Bool;
   "Module19Chanel11_DO" AT %Q289.2 : Bool;
   "Module19Chanel12_DO" AT %Q289.3 : Bool;
   "Module19Chanel13_DO" AT %Q289.4 : Bool;
   "Module19Chanel14_DO" AT %Q289.5 : Bool;
   "Module19Chanel15_DO" AT %Q289.6 : Bool;
   "Module19Chanel16_DO" AT %Q289.7 : Bool;
   "Module19Chanel1_AI" AT %IW288 : Int;
   "Module19Chanel2_AI" AT %IW290 : Int;
   "Module19Chanel3_AI" AT %IW292 : Int;
   "Module19Chanel4_AI" AT %IW294 : Int;
   "Module19Chanel5_AI" AT %IW296 : Int;
   "Module19Chanel6_AI" AT %IW298 : Int;
   "Module19Chanel7_AI" AT %IW300 : Int;
   "Module19Chanel8_AI" AT %IW302 : Int;
   "Module19Chanel1_AO" AT %QW288 : Int;
   "Module19Chanel2_AO" AT %QW290 : Int;
   "Module19Chanel3_AO" AT %QW292 : Int;
   "Module19Chanel4_AO" AT %QW294 : Int;
   "Module20Chanel1_DI" AT %I304.0 : Bool;
   "Module20Chanel2_DI" AT %I304.1 : Bool;
   "Module20Chanel3_DI" AT %I304.2 : Bool;
   "Module20Chanel4_DI" AT %I304.3 : Bool;
   "Module20Chanel5_DI" AT %I304.4 : Bool;
   "Module20Chanel6_DI" AT %I304.5 : Bool;
   "Module20Chanel7_DI" AT %I304.6 : Bool;
   "Module20Chanel8_DI" AT %I304.7 : Bool;
   "Module20Chanel9_DI" AT %I305.0 : Bool;
   "Module20Chanel10_DI" AT %I305.1 : Bool;
   "Module20Chanel11_DI" AT %I305.2 : Bool;
   "Module20Chanel12_DI" AT %I305.3 : Bool;
   "Module20Chanel13_DI" AT %I305.4 : Bool;
   "Module20Chanel14_DI" AT %I305.5 : Bool;
   "Module20Chanel15_DI" AT %I305.6 : Bool;
   "Module20Chanel16_DI" AT %I305.7 : Bool;
   "Module20Chanel1_DO" AT %Q304.0 : Bool;
   "Module20Chanel2_DO" AT %Q304.1 : Bool;
   "Module20Chanel3_DO" AT %Q304.2 : Bool;
   "Module20Chanel4_DO" AT %Q304.3 : Bool;
   "Module20Chanel5_DO" AT %Q304.4 : Bool;
   "Module20Chanel6_DO" AT %Q304.5 : Bool;
   "Module20Chanel7_DO" AT %Q304.6 : Bool;
   "Module20Chanel8_DO" AT %Q304.7 : Bool;
   "Module20Chanel9_DO" AT %Q305.0 : Bool;
   "Module20Chanel10_DO" AT %Q305.1 : Bool;
   "Module20Chanel11_DO" AT %Q305.2 : Bool;
   "Module20Chanel12_DO" AT %Q305.3 : Bool;
   "Module20Chanel13_DO" AT %Q305.4 : Bool;
   "Module20Chanel14_DO" AT %Q305.5 : Bool;
   "Module20Chanel15_DO" AT %Q305.6 : Bool;
   "Module20Chanel16_DO" AT %Q305.7 : Bool;
   "Module20Chanel1_AI" AT %IW304 : Int;
   "Module20Chanel2_AI" AT %IW306 : Int;
   "Module20Chanel3_AI" AT %IW308 : Int;
   "Module20Chanel4_AI" AT %IW310 : Int;
   "Module20Chanel5_AI" AT %IW312 : Int;
   "Module20Chanel6_AI" AT %IW314 : Int;
   "Module20Chanel7_AI" AT %IW316 : Int;
   "Module20Chanel8_AI" AT %IW318 : Int;
   "Module20Chanel1_AO" AT %QW304 : Int;
   "Module20Chanel2_AO" AT %QW306 : Int;
   "Module20Chanel3_AO" AT %QW308 : Int;
   "Module20Chanel4_AO" AT %QW310 : Int;
   "Module21Chanel1_DI" AT %I320.0 : Bool;
   "Module21Chanel2_DI" AT %I320.1 : Bool;
   "Module21Chanel3_DI" AT %I320.2 : Bool;
   "Module21Chanel4_DI" AT %I320.3 : Bool;
   "Module21Chanel5_DI" AT %I320.4 : Bool;
   "Module21Chanel6_DI" AT %I320.5 : Bool;
   "Module21Chanel7_DI" AT %I320.6 : Bool;
   "Module21Chanel8_DI" AT %I320.7 : Bool;
   "Module21Chanel9_DI" AT %I321.0 : Bool;
   "Module21Chanel10_DI" AT %I321.1 : Bool;
   "Module21Chanel11_DI" AT %I321.2 : Bool;
   "Module21Chanel12_DI" AT %I321.3 : Bool;
   "Module21Chanel13_DI" AT %I321.4 : Bool;
   "Module21Chanel14_DI" AT %I321.5 : Bool;
   "Module21Chanel15_DI" AT %I321.6 : Bool;
   "Module21Chanel16_DI" AT %I321.7 : Bool;
   "Module21Chanel1_DO" AT %Q320.0 : Bool;
   "Module21Chanel2_DO" AT %Q320.1 : Bool;
   "Module21Chanel3_DO" AT %Q320.2 : Bool;
   "Module21Chanel4_DO" AT %Q320.3 : Bool;
   "Module21Chanel5_DO" AT %Q320.4 : Bool;
   "Module21Chanel6_DO" AT %Q320.5 : Bool;
   "Module21Chanel7_DO" AT %Q320.6 : Bool;
   "Module21Chanel8_DO" AT %Q320.7 : Bool;
   "Module21Chanel9_DO" AT %Q321.0 : Bool;
   "Module21Chanel10_DO" AT %Q321.1 : Bool;
   "Module21Chanel11_DO" AT %Q321.2 : Bool;
   "Module21Chanel12_DO" AT %Q321.3 : Bool;
   "Module21Chanel13_DO" AT %Q321.4 : Bool;
   "Module21Chanel14_DO" AT %Q321.5 : Bool;
   "Module21Chanel15_DO" AT %Q321.6 : Bool;
   "Module21Chanel16_DO" AT %Q321.7 : Bool;
   "Module21Chanel1_AI" AT %IW320 : Int;
   "Module21Chanel2_AI" AT %IW322 : Int;
   "Module21Chanel3_AI" AT %IW324 : Int;
   "Module21Chanel4_AI" AT %IW326 : Int;
   "Module21Chanel5_AI" AT %IW328 : Int;
   "Module21Chanel6_AI" AT %IW330 : Int;
   "Module21Chanel7_AI" AT %IW332 : Int;
   "Module21Chanel8_AI" AT %IW334 : Int;
   "Module21Chanel1_AO" AT %QW320 : Int;
   "Module21Chanel2_AO" AT %QW322 : Int;
   "Module21Chanel3_AO" AT %QW324 : Int;
   "Module21Chanel4_AO" AT %QW326 : Int;
   "Module22Chanel1_DI" AT %I336.0 : Bool;
   "Module22Chanel2_DI" AT %I336.1 : Bool;
   "Module22Chanel3_DI" AT %I336.2 : Bool;
   "Module22Chanel4_DI" AT %I336.3 : Bool;
   "Module22Chanel5_DI" AT %I336.4 : Bool;
   "Module22Chanel6_DI" AT %I336.5 : Bool;
   "Module22Chanel7_DI" AT %I336.6 : Bool;
   "Module22Chanel8_DI" AT %I336.7 : Bool;
   "Module22Chanel9_DI" AT %I337.0 : Bool;
   "Module22Chanel10_DI" AT %I337.1 : Bool;
   "Module22Chanel11_DI" AT %I337.2 : Bool;
   "Module22Chanel12_DI" AT %I337.3 : Bool;
   "Module22Chanel13_DI" AT %I337.4 : Bool;
   "Module22Chanel14_DI" AT %I337.5 : Bool;
   "Module22Chanel15_DI" AT %I337.6 : Bool;
   "Module22Chanel16_DI" AT %I337.7 : Bool;
   "Module22Chanel1_DO" AT %Q336.0 : Bool;
   "Module22Chanel2_DO" AT %Q336.1 : Bool;
   "Module22Chanel3_DO" AT %Q336.2 : Bool;
   "Module22Chanel4_DO" AT %Q336.3 : Bool;
   "Module22Chanel5_DO" AT %Q336.4 : Bool;
   "Module22Chanel6_DO" AT %Q336.5 : Bool;
   "Module22Chanel7_DO" AT %Q336.6 : Bool;
   "Module22Chanel8_DO" AT %Q336.7 : Bool;
   "Module22Chanel9_DO" AT %Q337.0 : Bool;
   "Module22Chanel10_DO" AT %Q337.1 : Bool;
   "Module22Chanel11_DO" AT %Q337.2 : Bool;
   "Module22Chanel12_DO" AT %Q337.3 : Bool;
   "Module22Chanel13_DO" AT %Q337.4 : Bool;
   "Module22Chanel14_DO" AT %Q337.5 : Bool;
   "Module22Chanel15_DO" AT %Q337.6 : Bool;
   "Module22Chanel16_DO" AT %Q337.7 : Bool;
   "Module22Chanel1_AI" AT %IW336 : Int;
   "Module22Chanel2_AI" AT %IW338 : Int;
   "Module22Chanel3_AI" AT %IW340 : Int;
   "Module22Chanel4_AI" AT %IW342 : Int;
   "Module22Chanel5_AI" AT %IW344 : Int;
   "Module22Chanel6_AI" AT %IW346 : Int;
   "Module22Chanel7_AI" AT %IW348 : Int;
   "Module22Chanel8_AI" AT %IW350 : Int;
   "Module22Chanel1_AO" AT %QW336 : Int;
   "Module22Chanel2_AO" AT %QW338 : Int;
   "Module22Chanel3_AO" AT %QW340 : Int;
   "Module22Chanel4_AO" AT %QW342 : Int;
   "Module23Chanel1_DI" AT %I352.0 : Bool;
   "Module23Chanel2_DI" AT %I352.1 : Bool;
   "Module23Chanel3_DI" AT %I352.2 : Bool;
   "Module23Chanel4_DI" AT %I352.3 : Bool;
   "Module23Chanel5_DI" AT %I352.4 : Bool;
   "Module23Chanel6_DI" AT %I352.5 : Bool;
   "Module23Chanel7_DI" AT %I352.6 : Bool;
   "Module23Chanel8_DI" AT %I352.7 : Bool;
   "Module23Chanel9_DI" AT %I353.0 : Bool;
   "Module23Chanel10_DI" AT %I353.1 : Bool;
   "Module23Chanel11_DI" AT %I353.2 : Bool;
   "Module23Chanel12_DI" AT %I353.3 : Bool;
   "Module23Chanel13_DI" AT %I353.4 : Bool;
   "Module23Chanel14_DI" AT %I353.5 : Bool;
   "Module23Chanel15_DI" AT %I353.6 : Bool;
   "Module23Chanel16_DI" AT %I353.7 : Bool;
   "Module23Chanel1_DO" AT %Q352.0 : Bool;
   "Module23Chanel2_DO" AT %Q352.1 : Bool;
   "Module23Chanel3_DO" AT %Q352.2 : Bool;
   "Module23Chanel4_DO" AT %Q352.3 : Bool;
   "Module23Chanel5_DO" AT %Q352.4 : Bool;
   "Module23Chanel6_DO" AT %Q352.5 : Bool;
   "Module23Chanel7_DO" AT %Q352.6 : Bool;
   "Module23Chanel8_DO" AT %Q352.7 : Bool;
   "Module23Chanel9_DO" AT %Q353.0 : Bool;
   "Module23Chanel10_DO" AT %Q353.1 : Bool;
   "Module23Chanel11_DO" AT %Q353.2 : Bool;
   "Module23Chanel12_DO" AT %Q353.3 : Bool;
   "Module23Chanel13_DO" AT %Q353.4 : Bool;
   "Module23Chanel14_DO" AT %Q353.5 : Bool;
   "Module23Chanel15_DO" AT %Q353.6 : Bool;
   "Module23Chanel16_DO" AT %Q353.7 : Bool;
   "Module23Chanel1_AI" AT %IW352 : Int;
   "Module23Chanel2_AI" AT %IW354 : Int;
   "Module23Chanel3_AI" AT %IW356 : Int;
   "Module23Chanel4_AI" AT %IW358 : Int;
   "Module23Chanel5_AI" AT %IW360 : Int;
   "Module23Chanel6_AI" AT %IW362 : Int;
   "Module23Chanel7_AI" AT %IW364 : Int;
   "Module23Chanel8_AI" AT %IW366 : Int;
   "Module23Chanel1_AO" AT %QW352 : Int;
   "Module23Chanel2_AO" AT %QW354 : Int;
   "Module23Chanel3_AO" AT %QW356 : Int;
   "Module23Chanel4_AO" AT %QW358 : Int;
   "Module24Chanel1_DI" AT %I368.0 : Bool;
   "Module24Chanel2_DI" AT %I368.1 : Bool;
   "Module24Chanel3_DI" AT %I368.2 : Bool;
   "Module24Chanel4_DI" AT %I368.3 : Bool;
   "Module24Chanel5_DI" AT %I368.4 : Bool;
   "Module24Chanel6_DI" AT %I368.5 : Bool;
   "Module24Chanel7_DI" AT %I368.6 : Bool;
   "Module24Chanel8_DI" AT %I368.7 : Bool;
   "Module24Chanel9_DI" AT %I369.0 : Bool;
   "Module24Chanel10_DI" AT %I369.1 : Bool;
   "Module24Chanel11_DI" AT %I369.2 : Bool;
   "Module24Chanel12_DI" AT %I369.3 : Bool;
   "Module24Chanel13_DI" AT %I369.4 : Bool;
   "Module24Chanel14_DI" AT %I369.5 : Bool;
   "Module24Chanel15_DI" AT %I369.6 : Bool;
   "Module24Chanel16_DI" AT %I369.7 : Bool;
   "Module24Chanel1_DO" AT %Q368.0 : Bool;
   "Module24Chanel2_DO" AT %Q368.1 : Bool;
   "Module24Chanel3_DO" AT %Q368.2 : Bool;
   "Module24Chanel4_DO" AT %Q368.3 : Bool;
   "Module24Chanel5_DO" AT %Q368.4 : Bool;
   "Module24Chanel6_DO" AT %Q368.5 : Bool;
   "Module24Chanel7_DO" AT %Q368.6 : Bool;
   "Module24Chanel8_DO" AT %Q368.7 : Bool;
   "Module24Chanel9_DO" AT %Q369.0 : Bool;
   "Module24Chanel10_DO" AT %Q369.1 : Bool;
   "Module24Chanel11_DO" AT %Q369.2 : Bool;
   "Module24Chanel12_DO" AT %Q369.3 : Bool;
   "Module24Chanel13_DO" AT %Q369.4 : Bool;
   "Module24Chanel14_DO" AT %Q369.5 : Bool;
   "Module24Chanel15_DO" AT %Q369.6 : Bool;
   "Module24Chanel16_DO" AT %Q369.7 : Bool;
   "Module24Chanel1_AI" AT %IW368 : Int;
   "Module24Chanel2_AI" AT %IW370 : Int;
   "Module24Chanel3_AI" AT %IW372 : Int;
   "Module24Chanel4_AI" AT %IW374 : Int;
   "Module24Chanel5_AI" AT %IW376 : Int;
   "Module24Chanel6_AI" AT %IW378 : Int;
   "Module24Chanel7_AI" AT %IW380 : Int;
   "Module24Chanel8_AI" AT %IW382 : Int;
   "Module24Chanel1_AO" AT %QW368 : Int;
   "Module24Chanel2_AO" AT %QW370 : Int;
   "Module24Chanel3_AO" AT %QW372 : Int;
   "Module24Chanel4_AO" AT %QW374 : Int;
   "Module25Chanel1_DI" AT %I384.0 : Bool;
   "Module25Chanel2_DI" AT %I384.1 : Bool;
   "Module25Chanel3_DI" AT %I384.2 : Bool;
   "Module25Chanel4_DI" AT %I384.3 : Bool;
   "Module25Chanel5_DI" AT %I384.4 : Bool;
   "Module25Chanel6_DI" AT %I384.5 : Bool;
   "Module25Chanel7_DI" AT %I384.6 : Bool;
   "Module25Chanel8_DI" AT %I384.7 : Bool;
   "Module25Chanel9_DI" AT %I385.0 : Bool;
   "Module25Chanel10_DI" AT %I385.1 : Bool;
   "Module25Chanel11_DI" AT %I385.2 : Bool;
   "Module25Chanel12_DI" AT %I385.3 : Bool;
   "Module25Chanel13_DI" AT %I385.4 : Bool;
   "Module25Chanel14_DI" AT %I385.5 : Bool;
   "Module25Chanel15_DI" AT %I385.6 : Bool;
   "Module25Chanel16_DI" AT %I385.7 : Bool;
   "Module25Chanel1_DO" AT %Q384.0 : Bool;
   "Module25Chanel2_DO" AT %Q384.1 : Bool;
   "Module25Chanel3_DO" AT %Q384.2 : Bool;
   "Module25Chanel4_DO" AT %Q384.3 : Bool;
   "Module25Chanel5_DO" AT %Q384.4 : Bool;
   "Module25Chanel6_DO" AT %Q384.5 : Bool;
   "Module25Chanel7_DO" AT %Q384.6 : Bool;
   "Module25Chanel8_DO" AT %Q384.7 : Bool;
   "Module25Chanel9_DO" AT %Q385.0 : Bool;
   "Module25Chanel10_DO" AT %Q385.1 : Bool;
   "Module25Chanel11_DO" AT %Q385.2 : Bool;
   "Module25Chanel12_DO" AT %Q385.3 : Bool;
   "Module25Chanel13_DO" AT %Q385.4 : Bool;
   "Module25Chanel14_DO" AT %Q385.5 : Bool;
   "Module25Chanel15_DO" AT %Q385.6 : Bool;
   "Module25Chanel16_DO" AT %Q385.7 : Bool;
   "Module25Chanel1_AI" AT %IW384 : Int;
   "Module25Chanel2_AI" AT %IW386 : Int;
   "Module25Chanel3_AI" AT %IW388 : Int;
   "Module25Chanel4_AI" AT %IW390 : Int;
   "Module25Chanel5_AI" AT %IW392 : Int;
   "Module25Chanel6_AI" AT %IW394 : Int;
   "Module25Chanel7_AI" AT %IW396 : Int;
   "Module25Chanel8_AI" AT %IW398 : Int;
   "Module25Chanel1_AO" AT %QW384 : Int;
   "Module25Chanel2_AO" AT %QW386 : Int;
   "Module25Chanel3_AO" AT %QW388 : Int;
   "Module25Chanel4_AO" AT %QW390 : Int;
END_VAR

VAR_GLOBAL   // PLC tag table "Test_L"
   "dP_main" AT %MD100 : Real;
   "L_main" AT %MD104 : Real;
   "Current_main" AT %MD108 : Real;
   "dP_res" AT %MD112 : Real;
   "L_res" AT %MD116 : Real;
   "Current_res" AT %MD120 : Real;
END_VAR

VAR_GLOBAL   // PLC tag table "www"
   "retval" AT %MW400 : Int;
END_VAR

DATA_BLOCK "Q_gas"   // DB113
{ S7_Optimized_Access := 'FALSE' }
AUTHOR : Петров
VERSION : 0.1
// Расход газа (м3/ч)
// stored: InstanceOfName GAS_METER
"GAS_METER"
BEGIN
   impulse_N_module := 10;
   impulse_N_chanel := 16;
   scale_unit := 1000.0;
END_DATA_BLOCK

DATA_BLOCK "Alarm"   // DB151
{ S7_Optimized_Access := 'FALSE' }
VERSION : 0.1
   VAR
      Global_alarm : Bool;   // Обобщенный признак аварии
      Reset_alarms : Bool;   // Сброс аварий и предупреждений
      P_gas_before_BG_max : Bool;   // Повышение давления газа перед БГ
      P_gas_before_BG_min : Bool;   // Понижение давления газа перед БГ
      P_gas_before_burner_min : Bool;   // Понижение давления газа перед горелкой
      P_gas_before_burner_max : Bool;   // Повышение давления газа перед горелкой
      DS_off : Bool;   // Отключение ДС
      DV_off : Bool;   // Отключение ДВ
      dP_furnace_boiler_min : Bool;   // Понижение разряжения в топке
      P_air_before_burner_min : Bool;   // Понижение давления воздуха перед горелкой
      L_water_min : Bool;   // Понижение уровня воды в барабане
      L_water_max : Bool;   // Повышение уровня воды в барабане
      P_steam_max : Bool;   // Повышение давления пара в барабане
      Not_flame_burner : Bool;   // Невоспламенение или погасание факела горелки котла
      Alarm_stop_HMI : Bool;   // Нажата кнопка аварийного останова на панели оператора
      Alarm_stop_SCADA : Bool;   // Нажата кнопка аварийного останова на SCADA
      CO2 : Bool;   // СО2 порог 2
      CH4 : Bool;   // CH4
   END_VAR
BEGIN
END_DATA_BLOCK

DATA_BLOCK "Alarm_Enable"   // DB152
{ S7_Optimized_Access := 'FALSE' }
VERSION : 0.1
// Разрешение аварии
   VAR
      P_gas_before_BG_min : Bool;   // Понижение давления газа перед БГ
      P_gas_before_BG_max : Bool;   // Повышение давления газа перед БГ
      P_gas_before_burner_min : Bool;   // Понижение давления газа перед горелкой
      P_gas_before_burner_max : Bool;   // Повышение давления газа перед горелкой
      DS_off : Bool;   // Отключение ДС
      DV_off : Bool;   // Отключение ДВ
      dP_furnace_boiler_min : Bool;   // Понижение разряжения в топке
      P_air_before_burner_min : Bool;   // Понижение давления воздуха перед горелкой
      L_water_min : Bool;   // Понижение уровня воды в барабане
      L_water_max : Bool;   // Повышение уровня воды в барабане
      P_steam_max : Bool;   // Повышение давления пара в барабане
      Not_flame_burner : Bool;   // Невоспламенение или погасание факела горелки котла
      Alarm_stop_HMI : Bool := true;   // Нажата кнопка аварийного останова на панели оператора
      Alarm_stop_SCADA : Bool := true;   // Нажата кнопка аварийного останова на SCADA
      CO2 : Bool := true;   // СО2 порог 2
      CH4 : Bool := true;   // CH4
   END_VAR
BEGIN
END_DATA_BLOCK

DATA_BLOCK "Alarm_Timer"   // DB153
{ S7_Optimized_Access := 'FALSE' }
VERSION : 0.1
   VAR
      alarm_1_IN : Bool;
      alarm_1_Q : Bool;
      alarm_1_PT : Time;
      alarm_2_IN : Bool;
      alarm_2_Q : Bool;
      alarm_2_PT : Time;
      alarm_3_IN : Bool;
      alarm_3_Q : Bool;
      alarm_3_PT : Time;
      alarm_4_IN : Bool;
      alarm_4_Q : Bool;
      alarm_4_PT : Time;
      alarm_5_IN : Bool;
      alarm_5_Q : Bool;
      alarm_5_PT : Time;
      alarm_6_IN : Bool;
      alarm_6_Q : Bool;
      alarm_6_PT : Time;
      alarm_7_IN : Bool;
      alarm_7_Q : Bool;
      alarm_7_PT : Time;
      alarm_8_IN : Bool;
      alarm_8_Q : Bool;
      alarm_8_PT : Time;
      alarm_9_IN : Bool;
      alarm_9_Q : Bool;
      alarm_9_PT : Time;
      alarm_10_IN : Bool;
      alarm_10_Q : Bool;
      alarm_10_PT : Time;
      alarm_11_IN : Bool;
      alarm_11_Q : Bool;
      alarm_11_PT : Time;
      alarm_12_IN : Bool;
      alarm_12_Q : Bool;
      alarm_12_PT : Time;
      alarm_13_IN : Bool;
      alarm_13_Q : Bool;
      alarm_13_PT : Time;
      alarm_14_IN : Bool;
      alarm_14_Q : Bool;
      alarm_14_PT : Time;
      alarm_15_IN : Bool;
      alarm_15_Q : Bool;
      alarm_15_PT : Time;
      alarm_16_IN : Bool;
      alarm_16_Q : Bool;
      alarm_16_PT : Time;
      alarm_17_IN : Bool;
      alarm_17_Q : Bool;
      alarm_17_PT : Time;
   END_VAR
BEGIN
END_DATA_BLOCK

DATA_BLOCK "Warning"   // DB154
{ S7_Optimized_Access := 'FALSE' }
VERSION : 0.1
// Предупреждения
   VAR
      Sensor_T_water_before_economizer : Bool;   // Неисправность датчика Температуры питательной воды перед экономайзером
      Sensor_T_water_after_economizer : Bool;   // Неисправность датчика Температуры питательной воды после экономайзера
      Sensor_dP_water_boiler : Bool;   // Неисправность датчика Перепада давления питательной воды на котел
      Sensor_P_water_before_regul : Bool;   // Неисправность датчика Давления питательной воды до регулятора
      Sensor_P_water_after_regul : Bool;   // Неисправность датчика Давления питательной воды после регулятора
      Sensor_dP_steam : Bool;   // Неисправность датчика Перепада давления пара в магистраль
      Sensor_P_steam : Bool;   // Неисправность датчика Давления пара в барабане
      Sensor_dP_furnace_boiler : Bool;   // Неисправность датчика Разрежения в топке котла
      Sensor_P_gas_between_PZK1_and_PZK2 : Bool;   // Неисправность датчика Давления газа между ПЗК-1 и ПЗК-2
      Sensor_P_gas_before_burner : Bool;   // Неисправность датчика Давления газа перед горелкой
      Sensor_P_air_burner : Bool;   // Неисправность датчика Давления воздуха к горелке
      Sensor_ZRW_position : Bool;   // Неисправность датчика Положения рег. заслонки питательной воды на котел
      Sensor_ZRG_position : Bool;   // Неисправность датчика Положения рег. заслонки газа перед котлом
      Sensor_NAV_position : Bool;   // Неисправность датчика Положения направл. аппарата вентилятора
      Sensor_NAD_position : Bool;   // Неисправность датчика Положения направл. аппарата дымососа
      Sensor_T_exhaust_gas_before_economizer : Bool;   // Неисправность датчика Температуры уходящих дымовых газов перед экономайзером
      Sensor_T_exhaust_gas_after_economizer : Bool;   // Неисправность датчика Температуры уходящих дымовых газов после экономайзера
      Sensor_dP_exhaust_gas_before_economizer : Bool;   // Неисправность датчика Разрежения в дымоходе перед экономайзером
      Sensor_dP_exhaust_gas_after_economizer : Bool;   // Неисправность датчика Разрежения в дымоходе после экономайзера
      Sensor_L_water : Bool;   // Неисправность датчика Уровня воды в барабане
      Sensor_P_gas_before_BG : Bool;   // Неисправность датчика Давления газа перед БГ
      Sensor_T_gas_before_BG : Bool;   // Неисправность датчика Температуры газа перед БГ
      Sensor_P_steam_pipe : Bool;   // Неисправность датчика Давления пара в магистраль
      Sensor_T_steam : Bool;   // Неисправность датчика Температуры пара в магистраль
      Sensor_DV_current_frequency : Bool;   // Неисправность датчика Текущего значение частоты ПЧ вентилятора
      Sensor_DS_current_frequency : Bool;   // Неисправность датчика Текущего значение частоты ПЧ дымососа
      ZDSV_before_boiler_limit_rotational_moment : Bool;   // Сработал ограничитель крутящего момента ЗДСВ перед котлом
      GPZ_limit_rotational_moment : Bool;   // Сработал ограничитель крутящего момента ГПЗ
      Call_power_supply_cabinet : Bool;   // Вызов к шкафу электропитания
      DV_need_on_QF_invertor : Bool;   // ДВ. Необходимо включить QF ПЧ
      DV_need_on_QF_powergrid : Bool;   // ДВ. Необходимо включить QF Сети
      DV_no_voltage : Bool;   // ДВ. Неисправность напряжения в сети ШУД
      DS_need_on_QF_invertor : Bool;   // ДС. Необходимо включить QF ПЧ
      DS_need_on_QF_powergrid : Bool;   // ДС. Необходимо включить QF Сети
      DS_no_voltage : Bool;   // ДС. Неисправность напряжения в сети ШУД
      SHEU_no_voltage : Bool;   // Нет питания ШЭУ
      Power_PLC_from_UPS : Bool;   // Питание контроллера от ИБП
      UPS_Low_charge : Bool;   // Низкий заряд батареи ИБП
      ZRG_no_voltage : Bool;   // Нет питания ЗРГ
      ZDG_no_voltage : Bool;   // Нет питания ЗДГ
      NAV_no_voltage : Bool;   // Нет питания НАВ
      NAD_no_voltage : Bool;   // Нет питания НАД
      ZDSV_before_boiler_no_voltage : Bool;   // Нет питания ЗДСВ перед котлом
      GPZ_no_voltage : Bool;   // Нет питания ГПЗ
      ZRW_no_voltage : Bool;   // Нет питания ЗРВ
      DV_invertor_alarm : Bool;   // Авария ПЧ ДВ
      DS_invertor_alarm : Bool;   // Авария ПЧ ДС
      ZRG_manual : Bool;   // ЗРГ в местном режиме
      NAV_manual : Bool;   // НАВ в местном режиме
      NAD_manual : Bool;   // НАД в местном режиме
      DV_manual : Bool;   // ДВ в местном режиме
      DS_manual : Bool;   // ДС в местном режиме
      ZRW_manual : Bool;   // ЗРВ в местном режиме
      Not_flame_Igniter : Bool := false;   // Пламя запальника потухло
      PZK2_not_open : Bool := false;   // ПЗК2 не открылся
      P_water_min : Bool;   // Понижение давления сетевой воды
      L_water_min : Bool;   // Понижение уровня воды в барабане
      L_water_max : Bool;   // Повышение уровня воды в барабане
      P_steam_max : Bool;   // Повышение давления пара в барабане
      CO2 : Bool;   // СО2 порог 1
      dP_furnace_boiler_min : Bool;   // Понижение разряжения в топке
      P_air_before_burner_min : Bool;   // Понижение давления воздуха перед горелкой
      ZDG_not_close : Bool := false;   // ДГ не закрылся
      protection_block : Bool;   // Предупреждение. Имеется блокировка защиты
      Sensor_L_water_reserv : Bool;   // Неисправность резервного датчика Уровня воды в барабане
      Sensor_P_steam_reserv : Bool;   // Неисправность резервного датчика Давления пара в барабане
   END_VAR
BEGIN
END_DATA_BLOCK

DATA_BLOCK "Warning_Enable"   // DB155
{ S7_Optimized_Access := 'FALSE' }
VERSION : 0.1
// Разрешение предупреждения
   VAR
      Sensor_T_water_before_economizer : Bool := TRUE;   // Неисправность датчика Температуры питательной воды перед экономайзером
      Sensor_T_water_after_economizer : Bool := TRUE;   // Неисправность датчика Температуры питательной воды после экономайзера
      Sensor_dP_water_boiler : Bool := TRUE;   // Неисправность датчика Перепада давления питательной воды на котел
      Sensor_P_water_before_regul : Bool := TRUE;   // Неисправность датчика Давления питательной воды до регулятора
      Sensor_P_water_after_regul : Bool := TRUE;   // Неисправность датчика Давления питательной воды после регулятора
      Sensor_dP_steam : Bool := TRUE;   // Неисправность датчика Перепада давления пара в магистраль
      Sensor_P_steam : Bool := TRUE;   // Неисправность датчика Давления пара в барабане
      Sensor_dP_furnace_boiler : Bool := TRUE;   // Неисправность датчика Разрежения в топке котла
      Sensor_P_gas_between_PZK1_and_PZK2 : Bool := TRUE;   // Неисправность датчика Давления газа между ПЗК-1 и ПЗК-2
      Sensor_P_gas_before_burner : Bool := TRUE;   // Неисправность датчика Давления газа перед горелкой
      Sensor_P_air_burner : Bool := TRUE;   // Неисправность датчика Давления воздуха к горелке
      Sensor_ZRW_position : Bool := TRUE;   // Неисправность датчика Положения рег. заслонки питательной воды на котел
      Sensor_ZRG_position : Bool := TRUE;   // Неисправность датчика Положения рег. заслонки газа перед котлом
      Sensor_NAV_position : Bool := TRUE;   // Неисправность датчика Положения направл. аппарата вентилятора
      Sensor_NAD_position : Bool := TRUE;   // Неисправность датчика Положения направл. аппарата дымососа
      Sensor_T_exhaust_gas_before_economizer : Bool := TRUE;   // Неисправность датчика Температуры уходящих дымовых газов перед экономайзером
      Sensor_T_exhaust_gas_after_economizer : Bool := TRUE;   // Неисправность датчика Температуры уходящих дымовых газов после экономайзера
      Sensor_dP_exhaust_gas_before_economizer : Bool := TRUE;   // Неисправность датчика Разрежения в дымоходе перед экономайзером
      Sensor_dP_exhaust_gas_after_economizer : Bool := TRUE;   // Неисправность датчика Разрежения в дымоходе после экономайзера
      Sensor_L_water : Bool := TRUE;   // Неисправность датчика Уровня воды в барабане
      Sensor_P_gas_before_BG : Bool := TRUE;   // Неисправность датчика Давления газа перед БГ
      Sensor_T_gas_before_BG : Bool := TRUE;   // Неисправность датчика Температуры газа перед БГ
      Sensor_P_steam_pipe : Bool := TRUE;   // Неисправность датчика Давления пара в магистраль
      Sensor_T_steam : Bool := TRUE;   // Неисправность датчика Температуры пара в магистраль
      Sensor_DV_current_frequency : Bool := TRUE;   // Неисправность датчика Текущего значение частоты ПЧ вентилятора
      Sensor_DS_current_frequency : Bool := TRUE;   // Неисправность датчика Текущего значение частоты ПЧ дымососа
      ZDSV_before_boiler_limit_rotational_moment : Bool := TRUE;   // Сработал ограничитель крутящего момента ЗДСВ перед котлом
      GPZ_limit_rotational_moment : Bool := TRUE;   // Сработал ограничитель крутящего момента ГПЗ
      Call_power_supply_cabinet : Bool := TRUE;   // Вызов к шкафу электропитания
      DV_need_on_QF_invertor : Bool := TRUE;   // ДВ. Необходимо включить QF ПЧ
      DV_need_on_QF_powergrid : Bool := TRUE;   // ДВ. Необходимо включить QF Сети
      DV_no_voltage : Bool := TRUE;   // ДВ. Неисправность напряжения в сети ШУД
      DS_need_on_QF_invertor : Bool := TRUE;   // ДС. Необходимо включить QF ПЧ
      DS_need_on_QF_powergrid : Bool := TRUE;   // ДС. Необходимо включить QF Сети
      DS_no_voltage : Bool := TRUE;   // ДС. Неисправность напряжения в сети ШУД
      SHEU_no_voltage : Bool := TRUE;   // Нет питания ШЭУ
      Power_PLC_from_UPS : Bool := TRUE;   // Питание контроллера от ИБП
      UPS_Low_charge : Bool := TRUE;   // Низкий заряд батареи ИБП
      ZRG_no_voltage : Bool := TRUE;   // Нет питания ЗРГ
      ZDG_no_voltage : Bool := TRUE;   // Нет питания ЗДГ
      NAV_no_voltage : Bool := TRUE;   // Нет питания НАВ
      NAD_no_voltage : Bool := TRUE;   // Нет питания НАД
      ZDSV_before_boiler_no_voltage : Bool := TRUE;   // Нет питания ЗДСВ перед котлом
      GPZ_no_voltage : Bool := TRUE;   // Нет питания ГПЗ
      ZRW_no_voltage : Bool := TRUE;   // Нет питания ЗРВ
      DV_invertor_alarm : Bool := TRUE;   // Авария ПЧ ДВ
      DS_invertor_alarm : Bool := TRUE;   // Авария ПЧ ДС
      ZRG_manual : Bool := TRUE;   // ЗРГ в местном режиме
      NAV_manual : Bool := TRUE;   // НАВ в местном режиме
      NAD_manual : Bool := TRUE;   // НАД в местном режиме
      DV_manual : Bool := TRUE;   // ДВ в местном режиме
      DS_manual : Bool := TRUE;   // ДС в местном режиме
      ZRW_manual : Bool := TRUE;   // ЗРВ в местном режиме
      Not_flame_Igniter : Bool := TRUE;   // Пламя запальника потухло
      PZK2_not_open : Bool := TRUE;   // ПЗК2 не открылся
      P_water_min : Bool := TRUE;   // Понижение давления сетевой воды
      L_water_min : Bool := TRUE;   // Понижение уровня воды в барабане
      L_water_max : Bool := TRUE;   // Повышение уровня воды в барабане
      P_steam_max : Bool := TRUE;   // Повышение давления пара в барабане
      CO2 : Bool := TRUE;   // СО2 порог 1
      dP_furnace_boiler_min : Bool := TRUE;   // Понижение разряжения в топке
      P_air_before_burner_min : Bool := TRUE;   // Понижение давления воздуха перед горелкой
      ZDG_not_close : Bool := false;   // ЗДГ не закрылся
      Sensor_L_water_reserv : Bool := TRUE;   // Неисправность резервного датчика Уровня воды в барабане
      Sensor_P_steam_reserv : Bool := TRUE;   // Неисправность резервного датчика Давления пара в барабане
   END_VAR
BEGIN
END_DATA_BLOCK

DATA_BLOCK "Warning_Timer"   // DB156
{ S7_Optimized_Access := 'FALSE' }
VERSION : 0.1
   VAR
      warning_1_IN : Bool;
      warning_1_Q : Bool;
      warning_1_PT : Time;
      warning_2_IN : Bool;
      warning_2_Q : Bool;
      warning_2_PT : Time;
      warning_3_IN : Bool;
      warning_3_Q : Bool;
      warning_3_PT : Time;
      warning_4_IN : Bool;
      warning_4_Q : Bool;
      warning_4_PT : Time;
      warning_5_IN : Bool;
      warning_5_Q : Bool;
      warning_5_PT : Time;
      warning_6_IN : Bool;
      warning_6_Q : Bool;
      warning_6_PT : Time;
      warning_7_IN : Bool;
      warning_7_Q : Bool;
      warning_7_PT : Time;
      warning_8_IN : Bool;
      warning_8_Q : Bool;
      warning_8_PT : Time;
      warning_9_IN : Bool;
      warning_9_Q : Bool;
      warning_9_PT : Time;
      warning_10_IN : Bool;
      warning_10_Q : Bool;
      warning_10_PT : Time;
   END_VAR
BEGIN
END_DATA_BLOCK

DATA_BLOCK "Alarm_SP"   // DB174
{ S7_Optimized_Access := 'FALSE' }
VERSION : 0.1
// Аварийные уставки
   VAR
      TIME_P_gas_before_BG_max : Int := 5;   // Время формирования аварии. Повышение давления газа перед БГ (сек)
      TIME_P_gas_before_BG_min : Int := 5;   // Время формирования аварии. Понижение давления газа перед БГ (сек)
      P_gas_before_BG_max : Real := 28.0;   // Аварийная уставка. Высокое давление газа перед БГ
      P_gas_before_BG_min : Real := 20.0;   // Аварийная уставка. Низкое давление газа перед БГ
      TIME_P_gas_before_burner_min : Int := 5;   // Время формирования аварии. Понижение давления газа перед горелкой (сек)
      TIME_P_gas_before_burner_max : Int := 5;   // Время формирования аварии. Повышение давления газа перед горелкой (сек)
      P_gas_before_burner_max : Real := 20.0;   // Аварийная уставка. Высокое давление газа перед горелкой
      P_gas_before_burner_min : Real := 0.5;   // Аварийная уставка. Низкое давление газа перед горелкой
      TIME_DS_off : Int := 1;   // Время формирования аварии. Отключение ДС (сек)
      TIME_DV_off : Int := 1;   // Время формирования аварии. Отключение ДВ (сек)
      TIME_P_air_before_burner_min : Int := 5;   // Время формирования аварии. Понижение давления воздуха перед горелкой (сек)
      TIME_dP_furnace_boiler_min : Int := 15;   // Время формирования аварии. Понижение разряжения в топке (сек)
      dP_furnace_boiler_min : Real;   // Аварийная уставка. Низкое разрежение в топке
      P_air_before_burner_min : Real := 15.0;   // Аварийная уставка. Низкое давление воздуха перед горелкой
      TIME_L_water_min : Int := 1;   // Время формирования аварии. Понижение уровня воды в барабане (сек)
      TIME_L_water_max : Int := 5;   // Время формирования аварии. Повышение уровня воды в барабане (сек)
      L_water_min : Real := -150.0;   // Аварийная уставка. Низкий уровень воды в барабане
      L_water_max : Real := 150.0;   // Аварийная уставка. Высокий уровень воды в барабане
      TIME_P_steam_max : Int := 1;   // Время формирования аварии. Повышение давления пара в барабане (сек)
      P_steam_max : Real := 12.0;   // Аварийная уставка. Высокое давление пара в барабане
      TIME_Not_flame_burner : Int := 50;   // Время формирования аварии. Невоспламенение или погасание факела горелки котла (мсек)
      TIME_CO2 : Int := 5;   // Время формирования аварии. СО2 порог 2 (сек)
      TIME_CH4 : Int := 5;   // Время формирования аварии. CH4 (сек)
   END_VAR
BEGIN
END_DATA_BLOCK

DATA_BLOCK "Protections"   // DB175
{ S7_Optimized_Access := 'FALSE' }
VERSION : 0.1
// Защиты
   VAR
      Global : Bool;   // Сработка защиты
      P_gas_before_BG_max : Bool;   // Повышение давления газа перед БГ
      P_gas_before_BG_min : Bool;   // Понижение давления газа перед БГ
      P_gas_before_burner_min : Bool;   // Понижение давления газа перед горелкой
      P_gas_before_burner_max : Bool;   // Повышение давления газа перед горелкой
      DS_off : Bool;   // Отключение ДС
      DV_off : Bool;   // Отключение ДВ
      dP_in_furnance_min : Bool;   // Понижение разряжения в топке
      P_air_before_burner_min : Bool;   // Понижение давления воздуха перед горелкой
      L_water_min : Bool;   // Понижение уровня в барабане котла
      L_water_max : Bool;   // Повышение уровня в барабане котла
      P_steam_max : Bool;   // Повышение давления пара в барабане котла
      Not_flame_burner : Bool;   // Невоспламенение или погасание факела горелки котла
      Alarm_stop_HMI : Bool;   // Нажата кнопка аварийного останова на панели операторора
      Alarm_stop_SCADA : Bool;   // Нажата кнопка аварийного останова на SCADA
   END_VAR
BEGIN
END_DATA_BLOCK

DATA_BLOCK "Protections_BLOCK"   // DB176
{ S7_Optimized_Access := 'FALSE' }
VERSION : 0.1
// Блокировки защит
   VAR
      P_gas_before_BG_max : Bool;   // Повышение давления газа перед БГ
      P_gas_before_BG_min : Bool;   // Понижение давления газа перед БГ
      P_gas_before_burner_min : Bool;   // Понижение давления газа перед горелкой
      P_gas_before_burner_max : Bool;   // Повышение давления газа перед горелкой
      DS_off : Bool;   // Отключение ДС
      DV_off : Bool;   // Отключение ДВ
      dP_in_furnance_min : Bool;   // Понижение разряжения в топке
      P_air_before_burner_min : Bool;   // Понижение давления воздуха перед горелкой
      L_water_min : Bool;   // Понижение уровня в барабане котла
      L_water_max : Bool;   // Повышение уровня в барабане котла
      P_steam_max : Bool;   // Повышение давления пара в барабане котла
      Not_flame_burner : Bool;   // Невоспламенение или погасание факела горелки котла
      Alarm_stop_HMI : Bool;   // Нажата кнопка аварийного останова на панели операторора
      Alarm_stop_SCADA : Bool;   // Нажата кнопка аварийного останова на SCADA
   END_VAR
BEGIN
END_DATA_BLOCK

DATA_BLOCK "Warning_SP"   // DB179
{ S7_Optimized_Access := 'FALSE' }
VERSION : 0.1
// Предупредительные уставки
   VAR
      TIME_Not_flame_Igniter : Int := 300;   // Время формирования предупреждения. Пламя запальника потухло (мсек)
      TIME_PZK2_not_open : Int := 55;   // Время формирования предупреждения. ПЗК2 не открылся (сек)
      P_water_min : Real := 0.0;   // Низкое давление воды
      TIME_L_water_min : Int := 5;   // Время формирования предупреждения. Понижение уровня воды в барабане (сек)
      TIME_L_water_max : Int := 5;   // Время формирования предупреждения. Повышение уровня воды в барабане (сек)
      L_water_min : Real := -100.0;   // Низкий уровень воды в барабане
      L_water_max : Real := 100.0;   // Высокий уровень воды в барабане
      TIME_P_steam_max : Int := 0;   // Время формирования предупреждения. Повышение давления пара в барабане (сек)
      P_steam_max : Real := 10.0;   // Высокое давление пара в барабане
      TIME_ZDG_not_close : Int := 30;   // Время формирования предупреждения. ЗДГ не закрылся (сек)
   END_VAR
BEGIN
END_DATA_BLOCK

DATA_BLOCK "HMI"   // DB186
{ S7_Optimized_Access := 'FALSE' }
VERSION : 0.1
   VAR
      Btn_Ventilation_HMI : Bool;   // Кнопка ВЕНТИЛЯЦИЯ на панели оператора
      Btn_Ventilation_SCADA : Bool;   // Кнопка ВЕНТИЛЯЦИЯ на SCADA
      Btn_Ignition_HMI : Bool;   // Кнопка РОЗЖИГ на панели оператора
      Btn_Ignition_SCADA : Bool;   // Кнопка РОЗЖИГ на SCADA
      Btn_normal_stop_HMI : Bool;   // Кнопка НОРМАЛЬНЫЙ ОСТАНОВ на панели оператора
      Btn_normal_stop_SCADA : Bool;   // Кнопка НОРМАЛЬНЫЙ ОСТАНОВ на SCADA
      Btn_alarm_stop_HMI : Bool;   // Кнопка АВАРИЙНЫЙ ОСТАНОВ на панели оператора
      Btn_alarm_stop_SCADA : Bool;   // Кнопка АВАРИЙНЫЙ ОСТАНОВ на SCADA
      Btn_test_press_HMI : Bool;   // Кнопка ТЕСТОВАЯ ОПРЕССОВКА на панели оператора
      Btn_test_ignition_HMI : Bool;   // Кнопка ТЕСТОВЫЙ РОЗЖИГ на панели оператора
      Btn_manual_ignition_HMI : Bool;   // Кнопка Ручной РОЗЖИГ на панели оператора
      Btn_reset_sound_HMI : Bool;   // Кнопка СБРОС ЗВУКА на панели оператора
      Btn_Ventilation_HMI_Log : Bool;   // Кнопка ВЕНТИЛЯЦИЯ на панели оператора для журнала событий
      Btn_Ventilation_SCADA_Log : Bool;   // Кнопка ВЕНТИЛЯЦИЯ на SCADA для журнала событий
      Btn_Ventilation_ShAU_Log : Bool;   // Кнопка ВЕНТИЛЯЦИЯ на ШАУ для журнала событий
      Btn_Ignition_HMI_Log : Bool;   // Кнопка РОЗЖИГ на панели оператора для журнала событий
      Btn_Ignition_SCADA_Log : Bool;   // Кнопка РОЗЖИГ на SCADA для журнала событий
      Btn_Ignition_ShAU_Log : Bool;   // Кнопка РОЗЖИГ на ШАУ для журнала событий
      Btn_normal_stop_HMI_Log : Bool;   // Кнопка НОРМАЛЬНЫЙ ОСТАНОВ на панели оператора для журнала событий
      Btn_normal_stop_SCADA_Log : Bool;   // Кнопка НОРМАЛЬНЫЙ ОСТАНОВ на SCADA для журнала событий
      Btn_alarm_stop_HMI_Log : Bool;   // Кнопка АВАРИЙНЫЙ ОСТАНОВ на панели оператора для журнала событий
      Btn_alarm_stop_SCADA_Log : Bool;   // Кнопка АВАРИЙНЫЙ ОСТАНОВ на SCADA для журнала событий
      Btn_emergency_stop_ShAU_Log : Bool;   // Кнопка ЭКСТРЕННЫЙ ОСТАНОВ на ШАУ для журнала событий
      Btn_test_press_HMI_Log : Bool;   // Кнопка ТЕСТОВАЯ ОПРЕССОВКА на панели оператора для журнала событий
      Btn_test_ignition_HMI_Log : Bool;   // Кнопка ТЕСТОВЫЙ РОЗЖИГ на панели оператора для журнала событий
      Btn_manual_ignition_HMI_Log : Bool;   // Кнопка Ручной РОЗЖИГ на панели оператора для журнала событий
      Btn_reset_sound_HMI_Log : Bool;   // Кнопка СБРОС ЗВУКА на панели оператора для журнала событий
      Btn_reset_alarms_ShAU_Log : Bool;   // Сброс аварий на ШАУ для журнала событий
      Reset_alarms_Log : Bool;   // Сброс аварий для журнала событий
      RegMap_Apply_Log : Bool;   // Режимная карта. Применить. Для журнала событий
      DS_Manual_Start_Log : Bool;   // ДС. Ручное управление. Пуск. Для журнала событий
      DS_Manual_Stop_Log : Bool;   // ДС. Ручное управление. Стоп. Для журнала событий
      DV_Manual_Start_Log : Bool;   // ДВ. Ручное управление. Пуск. Для журнала событий
      DV_Manual_Stop_Log : Bool;   // ДВ. Ручное управление. Стоп. Для журнала событий
      ZDG_Manual_open_Log : Bool;   // ЗДГ. Ручное управление. Открыть. Для журнала событий
      ZDG_Manual_close_Log : Bool;   // ЗДГ. Ручное управление. Закрыть. Для журнала событий
      ZDG_Manual_stop_Log : Bool;   // ЗДГ. Ручное управление. Стоп. Для журнала событий
      GPZ_Manual_open_Log : Bool;   // ЗДГ. Ручное управление. Открыть. Для журнала событий
      GPZ_Manual_close_Log : Bool;   // ЗДГ. Ручное управление. Закрыть. Для журнала событий
      GPZ_Manual_stop_Log : Bool;   // ЗДГ. Ручное управление. Стоп. Для журнала событий
      ZDSV_before_boiler_Manual_open_Log : Bool;   // ЗДСВ перед котлом. Ручное управление. Открыть. Для журнала событий
      ZDSV_before_boiler_Manual_close_Log : Bool;   // ЗДСВ перед котлом. Ручное управление. Закрыть. Для журнала событий
      ZDSV_before_boiler_Manual_stop_Log : Bool;   // ЗДСВ перед котлом. Ручное управление. Стоп. Для журнала событий
      Current_SP_P_air : Real;   // Текущая уставка регулятора давления воздуха
      Current_SP_dP_furnance : Real;   // Текущая уставка регулятора разрежения
      TIME_converter_minute : Int;
      TIME_converter_second : Int;
      LTIME_converter_day : DInt;
      LTIME_converter_hour : Int;
      INDICATION_TIME_1 : USInt;
      INDICATION_TIME_2 : USInt;
      TIME_converter_IN : Time;
      LTIME_converter_IN : LTime;
   END_VAR
BEGIN
END_DATA_BLOCK

DATA_BLOCK "FRONT"   // DB203
{ S7_Optimized_Access := 'FALSE' }
VERSION : 0.1
   VAR
      Alarm_1 : Bool;   // Фронт аварии1
      Alarm_2 : Bool;   // Фронт аварии2
      Alarm_3 : Bool;   // Фронт аварии3
      Alarm_4 : Bool;   // Фронт аварии4
      Alarm_5 : Bool;   // Фронт аварии5
      Alarm_6 : Bool;   // Фронт аварии6
      Alarm_7 : Bool;   // Фронт аварии7
      Alarm_8 : Bool;   // Фронт аварии8
      Alarm_9 : Bool;   // Фронт аварии9
      Alarm_10 : Bool;   // Фронт аварии10
      Alarm_11 : Bool;   // Фронт аварии11
      Alarm_12 : Bool;   // Фронт аварии12
      Alarm_13 : Bool;   // Фронт аварии13
      Alarm_14 : Bool;   // Фронт аварии14
      Alarm_15 : Bool;   // Фронт аварии15
      Alarm_16 : Bool;   // Фронт аварии16
      Btn_Ventilation_HMI : Bool;   // Фронт нажатия кнопки ВЕНТИЛЯЦИЯ на HMI
      Btn_Ventilation_SCADA : Bool;   // Фронт нажатия кнопки ВЕНТИЛЯЦИЯ на SCADA
      Btn_Ignition_HMI : Bool;   // Фронт нажатия кнопки РОЗЖИГ на HMI
      Btn_Ignition_SCADA : Bool;   // Фронт нажатия кнопки РОЗЖИГ на SCADA
      Btn_Normal_stop_HMI : Bool;   // Фронт нажатия кнопки НОРМАЛЬНЫЙ ОСТАНОВ на HMI
      Btn_Normal_stop_SCADA : Bool;   // Фронт нажатия кнопки НОРМАЛЬНЫЙ ОСТАНОВ на SCADA
      Btn_Alarm_stop_HMI : Bool;   // Фронт нажатия кнопки АВАРИЙНЫЙ ОСТАНОВ на HMI
      Btn_Alarm_stop_SCADA : Bool;   // Фронт нажатия кнопки АВАРИЙНЫЙ ОСТАНОВ на SCADA
      Btn_test_press_HMI : Bool;   // Фронт нажатия кнопки ТЕСТОВАЯ ОПРЕССОВКА на HMI
      Btn_test_ignition_HMI : Bool;   // Фронт нажатия кнопки ТЕСТОВЫЙ РОЗЖИГ на HMI
      Btn_manual_ignition_HMI : Bool;   // Фронт нажатия кнопки РУЧНОЙ РОЗЖИГ на HMI
      Btn_reset_sound_HMI : Bool;   // Фронт нажатия кнопки СБРОС ЗВУКА на HMI
      DS_mode : Bool;   // Фронт перевода ДС в ручной режим
      DV_mode : Bool;   // Фронт перевода ДВ в ручной режим
      IVN_mode : Bool;   // Фронт перевода ИВН в ручной режим
      KB_mode : Bool;   // Фронт перевода КБ в ручной режим
      KO_mode : Bool;   // Фронт перевода КО в ручной режим
      KZ_mode : Bool;   // Фронт перевода КЗ в ручной режим
      PZK1_mode : Bool;   // Фронт перевода ПЗК1 в ручной режим
      PZK2_mode : Bool;   // Фронт перевода ПЗК2 в ручной режим
   END_VAR
BEGIN
END_DATA_BLOCK

DATA_BLOCK "Timer"   // DB204
{ S7_Optimized_Access := 'FALSE' }
VERSION : 0.1
   VAR
      test_sound_IN : Bool;
      test_sound_Q : Bool;
      test_sound_PT : Time;
      protection_13_IN : Bool;
      protection_13_Q : Bool;
      protection_13_PT : Time;
      Log_IN : Bool;
      Log_Q : Bool;
      Log_PT : Time := T#1s500ms;
      IGNITION_temp_IN : Bool;
      IGNITION_temp_Q : Bool;
      IGNITION_temp_PT : Time;
      IGNITION_control_flame_IN : Bool;
      IGNITION_control_flame_Q : Bool;
      IGNITION_control_flame_PT : Time;
      PRESS_temp_IN : Bool;
      PRESS_temp_Q : Bool;
      PRESS_temp_PT : Time;
      VENTILATION_temp_IN : Bool;
      VENTILATION_temp_Q : Bool;
      VENTILATION_temp_PT : Time;
      VENTILATION_IN : Bool;
      VENTILATION_R : Bool;
      VENTILATION_Q : Bool;
      VENTILATION_PT : Time;
      MIN_POWER_temp_IN : Bool;
      MIN_POWER_temp_Q : Bool;
      MIN_POWER_temp_PT : Time;
      MIN_POWER_1_IN : Bool;
      MIN_POWER_1_Q : Bool;
      MIN_POWER_1_PT : Time;
      MIN_POWER_2_IN : Bool;
      MIN_POWER_2_Q : Bool;
      MIN_POWER_2_PT : Time;
      HEATING_temp_IN : Bool;
      HEATING_temp_Q : Bool;
      HEATING_temp_PT : Time;
      STOP_PRESS_temp_IN : Bool;
      STOP_PRESS_temp_Q : Bool;
      STOP_PRESS_temp_PT : Time;
      SHORT_VENTILATION_temp_IN : Bool;
      SHORT_VENTILATION_temp_Q : Bool;
      SHORT_VENTILATION_temp_PT : Time;
      EMERGENCY_STOP_temp_IN : Bool;
      EMERGENCY_STOP_temp_Q : Bool;
      EMERGENCY_STOP_temp_PT : Time;
      ALARM_STOP_temp_IN : Bool;
      ALARM_STOP_temp_Q : Bool;
      ALARM_STOP_temp_PT : Time;
      PLAN_STOP_temp_IN : Bool;
      PLAN_STOP_temp_Q : Bool;
      PLAN_STOP_temp_PT : Time;
      RUN_temp_IN : Bool;
      RUN_temp_Q : Bool;
      RUN_temp_PT : LTime;
      close_KZ_IN : Bool;
      close_KZ_Q : Bool;
      close_KZ_PT : Time;
      avto_reset_IVN_IN : Bool;
      avto_reset_IVN_Q : Bool;
      avto_reset_IVN_PT : Time;
      IND_1_IN : Bool;
      IND_1_Q : Bool;
      IND_1_PT : Time;
      IND_2_IN : Bool;
      IND_2_Q : Bool;
      IND_2_PT : Time;
      STOP_MIN_POWER_1_IN : Bool;
      STOP_MIN_POWER_1_Q : Bool;
      STOP_MIN_POWER_1_PT : Time;
      STOP_MIN_POWER_2_IN : Bool;
      STOP_MIN_POWER_2_Q : Bool;
      STOP_MIN_POWER_2_PT : Time;
      Close_GPZ_IN : Bool;
      Close_GPZ_Q : Bool;
      Close_GPZ_PT : Time;
   END_VAR
BEGIN
END_DATA_BLOCK

DATA_BLOCK "Technology"   // DB221
{ S7_Optimized_Access := 'FALSE' }
VERSION : 0.1
   VAR
      Regim : USInt;   // Текущий режим работы
      Regim_off_step : USInt;   // Режим ОТКЛ. Текущий шаг
      Regim_check_step : USInt;   // Режим ПРОВЕРКА. Текущий шаг
      Regim_ventilation_step : USInt;   // Режим ВЕНТИЛЯЦИЯ. Текущий шаг
      Regim_press_step : USInt;   // Режим ОПРЕССОВКА. Текущий шаг
      Regim_ignition_step : USInt;   // Режим РОЗЖИГ. Текущий шаг
      Regim_min_power_step : USInt;   // Режим ВЫХОД НА МИН МОЩНОСТЬ. Текущий шаг
      Regim_heating_step : USInt;   // Режим ПРОГРЕВ. Текущий шаг
      Regim_run_step : USInt;   // Режим РАБОТА. Текущий шаг
      Regim_emergency_stop_step : USInt;   // Режим ЭКСТРЕННЫЙ ОСТАНОВ. Текущий шаг
      Regim_alarm_stop_step : USInt;   // Режим АВАРИЙНЫЙ ОСТАНОВ. Текущий шаг
      Regim_plan_stop_step : USInt;   // Режим ПЛАНОВЫЙ ОСТАНОВ. Текущий шаг
      Regim_stop_press_step : USInt;   // Режим ПОСТОСТАНОВОЧНАЯ ОПРЕССОВКА. Текущий шаг
      Regim_short_ventilation_step : USInt;   // Режим УКОРОЧЕННАЯ ВЕНТИЛЯЦИЯ. Текущий шаг
      Regim_test_press_step : USInt;   // Режим ТЕСТОВАЯ ОПРЕССОВКА. Текущий шаг
      Regim_test_ignition_step : USInt;   // Режим ТЕСТОВЫЙ РОЗЖИГ. Текущий шаг
      Ventilation_conducted : Bool;   // Вентиляция проведена
      Test_press_run : Bool;   // Запущена тестовая опрессовка
      Short_ventilation_enable : Bool := true;   // Разрешение проведения УКОРОЧЕННОЙ ВЕНТИЛЯЦИИ
      Test_ignition_run : Bool;   // Запущен тестовый розжиг
      Substage : Int;   // Подрежим
      transition_ignition : Bool;   // Был переход в розжиг и откытие ПЗК2
      SP_L_water : Real := 65.0;   // Уставка уровня воды в барабане
      SP_P_steam : Real := 5.8;   // Уставка давления пара в барабане
      SP_TIME_Ventilation : Int := 600;   // Уставка времени вентиляции топки перед розжигом (сек)
      SP_TIME_Ventilation_start : Int := 10;   // Уставка времени определения начала вентиляции (сек)
      DB_P_air_ventilation : Int := 15;   // Допустимое отклонение P воздуха при вентиляции (%)
      DB_dP_furnace_ventilation : Int := 15;   // Допустимое отклонение разрежения в топке при вентиляции (%)
      DB_P_air_ignition : Int := 10;   // Допустимое отклонение P воздуха при розжиге (%)
      DB_dP_furnace_ignition : Int := 20;   // Допустимое отклонение разряжения в топке при розжиге (%)
      SP_TIME_check_P_between_PZK : Int := 9;   // Уставка времени проверки давления между ПЗК при опрессовке (сек)
      SP_P_between_PZK_check_max : Real := 20.0;   // Уставка MAX Давления между ПЗК при опрессовке
      SP_P_between_PZK_check_min : Real := 3.0;   // Уставка времени вентиляции топки перед розжигом (сек)
      CNT_Igniter : Int;   // Счетчик попыток розжига запальника
      Heating_enable : Bool := true;   // Разрешение режима ПРОГРЕВ
      Max_P_gas_heating : Real := 1.2;   // Max давления газа для режима прогрев
      SP_TIME_Heating : Int := 3;   // Уставка времени прогрева (мин)
      SP_T_water_after_boiler : Real := 72.0;   // Уставка Т воды после котла
      Stop_press_enable : Bool := true;   // Разрешение режима ПОСТОСТАНОВОЧНАЯ ОПРЕССОВКА
      SP_TIME_check_P_stop_press_min : Int := 5;   // Уставка времени проверки давления между ПЗК на min при постостановочной опрессовке (сек)
      SP_TIME_check_P_stop_press_max : Int := 5;   // Уставка времени проверки давления между ПЗК на max при постостановочной опрессовке (сек)
      SP_TIME_Short_ventilation : Int := 120;   // Уставка времени укороченной вентиляции топки (сек)
      Q_gas_scale_unit : Int := 100;   // Цена одного импульса (литр)
      P_atm : Real := 0.101325;   // Атмочферное давление (Мпа)
      K_gas : Real := 1.0;   // Коэффициент сжимаемости газа
      SP_TIME_MIN_power_ZRG_drive : Int := 350;   // Уставка времени движения ЗРГ при выходе на минимальную мощность (мсек)
      SP_TIME_MIN_power_ZRG_stop : Int := 4000;   // Уставка времени останова ЗРГ при выходе на минимальную мощность (мсек)
      Offset_level_water : Real;   // Смещение уровня воды (мм)
   END_VAR
BEGIN
END_DATA_BLOCK

DATA_BLOCK "TIME_converter_DB"   // DB222
{ S7_Optimized_Access := 'FALSE' }
VERSION : 0.1
// stored: InstanceOfName TIME_converter
"TIME_converter"
BEGIN
END_DATA_BLOCK

DATA_BLOCK "LTIME_converter_DB"   // DB223
{ S7_Optimized_Access := 'FALSE' }
VERSION : 0.1
// stored: InstanceOfName LTIME_converter
"LTIME_converter"
BEGIN
END_DATA_BLOCK

DATA_BLOCK "PID_impulse_ZRG_DB"   // DB224
{ S7_Optimized_Access := 'FALSE' }
VERSION : 0.1
// stored: InstanceOfName PID_impulse
"PID_impulse"
BEGIN
END_DATA_BLOCK

DATA_BLOCK "RT_INFO_DB"   // DB240
{ S7_Optimized_Access := 'FALSE' }
VERSION : 0.1
   VAR
      INFO : LTime;
      Ret_val : Int;
      Cycle : UDInt;   // Текущее время цикла (мс)
      temp : UDInt;
   END_VAR
BEGIN
END_DATA_BLOCK

DATA_BLOCK "RegMap"   // DB241
{ S7_Optimized_Access := 'FALSE' }
VERSION : 0.1
   VAR
      P_gaz_1 : Real := 1.1;   // P газа 1 точка
      P_gaz_2 : Real := 3.0;   // P газа 2 точка
      P_gaz_3 : Real := 4.0;   // P газа 3 точка
      P_gaz_4 : Real := 5.04;   // P газа 4 точка
      P_gaz_5 : Real := 7.0;   // P газа 5 точка
      P_gaz_6 : Real := 10.0;   // P газа 6 точка
      P_gaz_7 : Real := 10.1;   // P газа 7 точка
      P_gaz_8 : Real := 10.2;   // P газа 8 точка
      P_air_ventilation : Real := 250.0;   // Р воздуха Вентиляция
      P_air_ignition : Real := 50.0;   // Р воздуха Розжиг
      P_air_1 : Real := 50.0;   // Р воздуха 1 точка
      P_air_2 : Real := 75.0;   // Р воздуха 2 точка
      P_air_3 : Real := 130.0;   // Р воздуха 3 точка
      P_air_4 : Real := 190.0;   // Р воздуха 4 точка
      P_air_5 : Real := 330.0;   // Р воздуха 5 точка
      P_air_6 : Real := 570.0;   // Р воздуха 6 точка
      P_air_7 : Real := 570.0;   // Р воздуха 7 точка
      P_air_8 : Real := 570.0;   // Р воздуха 8 точка
      dP_furnace_ventilation : Real := -30.0;   // dP в топке Вентиляция
      dP_furnace_ignition : Real := -30.0;   // dP в топке Розжиг
      dP_furnace_1 : Real := -30.0;   // dP в топке 1 точка
      dP_furnace_2 : Real := -30.0;   // dP в топке 2 точка
      dP_furnace_3 : Real := -30.0;   // dP в топке 3 точка
      dP_furnace_4 : Real := -30.0;   // dP в топке 4 точка
      dP_furnace_5 : Real := -30.0;   // dP в топке 5 точка
      dP_furnace_6 : Real := -30.0;   // dP в топке 6 точка
      dP_furnace_7 : Real := -30.0;   // dP в топке 7 точка
      dP_furnace_8 : Real := -30.0;   // dP в топке 8 точка
      P_air_regim_map : Real := 0.002893518;   // Р воздуха по режимной карте
      dP_furnace_regim_map : Real := 0.002893518;   // dP в топке по режимной карте
      Apply : Bool := FALSE;   // Применить
      Error : Bool := TRUE;   // Ошибка
      Reset : Bool := FALSE;   // Сброс
   END_VAR
BEGIN
END_DATA_BLOCK

DATA_BLOCK "Message"   // DB242
{ S7_Optimized_Access := 'FALSE' }
VERSION : 0.1
   VAR
      OFF_Waiting_btn_ventilation : Bool;   // ОТКЛ. Ожидание нажатия кнопки ВЕНТИЛЯЦИЯ
      OFF_Param_ventilation_not_norm : Bool;   // ОТКЛ. Параметры вентиляции не в норме
      VENTILATION_not_initial_state_gas : Bool;   // ВЕНТИЛЯЦИЯ. Механизмы по газу не переведены в исходное состояние
      VENTILATION_DS_need_dist_mode : Bool;   // ВЕНТИЛЯЦИЯ. Необходимо перевести ДС в дистанционный режим
      VENTILATION_DV_need_dist_mode : Bool;   // ВЕНТИЛЯЦИЯ. Необходимо перевести ДВ в дистанционный режим
      VENTILATION_not_initial_state_air : Bool;   // ВЕНТИЛЯЦИЯ. Механизмы по воздуху не переведены в исходное состояние
      VENTILATION_NAV_not_close : Bool;   // ВЕНТИЛЯЦИЯ. НАВ не закрылись
      VENTILATION_NAD_not_open : Bool;   // ВЕНТИЛЯЦИЯ. НАД не открылись
      VENTILATION_NAV_or_NAD_not_open : Bool;   // ВЕНТИЛЯЦИЯ. НАВ или НАД не открылись
      VENTILATION_DS_not_on : Bool;   // ВЕНТИЛЯЦИЯ. ДС не включился
      VENTILATION_DV_not_on : Bool;   // ВЕНТИЛЯЦИЯ. ДВ не включился
      VENTILATION_run : Bool;   // ВЕНТИЛЯЦИЯ. Идет вентиляция топки
      VENTILATION_not : Bool;   // ВЕНТИЛЯЦИЯ. Нет вентиляции топки
      VENTILATION_alarm : Bool;   // ВЕНТИЛЯЦИЯ. Вентиляция не выполнена
      VENTILATION_ok : Bool;   // ВЕНТИЛЯЦИЯ. Вентиляция успешно проведена
      VENTILATION_Check_param : Bool;   // ВЕНТИЛЯЦИЯ. Проверьте параметры вентиляции
      VENTILATION_NAD_not_open_manual : Bool;   // ВЕНТИЛЯЦИЯ. НАД в местном режиме и не открыты
      VENTILATION_NAV_not_open_manual : Bool;   // ВЕНТИЛЯЦИЯ. НАВ в местном режиме и не открыты
      PRESS_not_initial_state_gas : Bool;   // ОПРЕССОВКА. Механизмы по газу не переведены в исходное состояние
      PRESS_ZRG_not_close : Bool;   // ОПРЕССОВКА. ЗРГ не закрылся
      PRESS_ZDG_not_open : Bool;   // ОПРЕССОВКА. ЗДГ не открылся
      PRESS_P_before_BG_alarm : Bool;   // ОПРЕССОВКА. Давление до БГ не в норме, Устраните неисправность и для продолжения нажмите кн. Розжиг
      PRESS_PZK1_or_KO_untight : Bool;   // ОПРЕССОВКА. ПЗК1 или КО негерметичен
      PRESS_Not_orifice_plate_or_PZK1_untight : Bool;   // ОПРЕССОВКА. Нет дроссельной шайбы или ПЗК1 негерметичен
      PRESS_PZK2_or_KB_untight : Bool;   // ОПРЕССОВКА. ПЗК2 или КБ негерметичен
      TEST_PRESS_ok : Bool;   // ТЕСТОВАЯ ОПРЕССОВКА. Прошла успешно
      IGNITION_Not_flame_igniter : Bool;   // РОЗЖИГ. Нет пламени запальника
      IGNITION_Flame_burner_OK : Bool;   // РОЗЖИГ. Есть пламя горелки
      IGNITION_ZRG_not_close : Bool;   // РОЗЖИГ. ЗРГ не закрыт
      IGNITION_PZK2_not_close : Bool;   // РОЗЖИГ. ПЗК2 не закрыт
      IGNITION_KZ_not_close : Bool;   // РОЗЖИГ. КЗ не закрыт
      IGNITION_KB_not_close : Bool;   // РОЗЖИГ. КБ не закрылся
      IGNITION_PZK1_not_open : Bool;   // РОЗЖИГ. ПЗК1 не открылся
      IGNITION_KZ_not_open : Bool;   // РОЗЖИГ. КЗ не открылся
      IGNITION_not_initial_state_gas : Bool;   // РОЗЖИГ. Механизмы по газу не переведены в исходное состояние
      TEST_IGNITION_ok : Bool;   // ТЕСТОВЫЙ РОЗЖИГ. Прошел успешно
      EMERGENCY_STOP_not_initial_state : Bool;   // ЭКСТРЕННЫЙ ОСТАНОВ. Устройства не переведены в исходное состояние
      ALARM_STOP_not_initial_state_gas : Bool;   // АВАРИЙНЫЙ ОСТАНОВ. Механизмы по газу не переведены в исходное состояние
      PLAN_STOP_not_initial_state_gas : Bool;   // ПЛАНОВЫЙ ОСТАНОВ. Механизмы по газу не переведены в исходное состояние
      STOP_PRESS_P_before_BG_min : Bool;   // ПОСТОСТАНОВОЧНАЯ ОПРЕССОВКА. Давление до БГ низкое
      STOP_PRESS_PZK1_or_KO_untight : Bool;   // ПОСТОСТАНОВОЧНАЯ ОПРЕССОВКА. ПЗК1 или КО негерметичен
      STOP_PRESS_PZK2_or_KB_untight : Bool;   // ПОСТОСТАНОВОЧНАЯ ОПРЕССОВКА. ПЗК2 или КБ негерметичен
      STOP_PRESS_success : Bool;   // ПОСТОСТАНОВОЧНАЯ ОПРЕССОВКА. Успешно проведена
      SHORT_VENTILATION_ok : Bool;   // УКОРОЧЕННАЯ ВЕНТИЛЯЦИЯ. проведена
      VENTILATION_BRU_NAD_need_avto_mode : Bool;   // ВЕНТИЛЯЦИЯ. Необходимо перевести БРУ НАД в автоматический режим
      VENTILATION_BRU_NAV_need_avto_mode : Bool;   // ВЕНТИЛЯЦИЯ. Необходимо перевести БРУ НАВ в автоматический режим
   END_VAR
BEGIN
END_DATA_BLOCK

DATA_BLOCK "Engineering_units"   // DB244
{ S7_Optimized_Access := 'FALSE' }
VERSION : 0.1
   VAR
      pressure_01_EU : Word := 3;
      pressure_02_EU : Word := 2;
      pressure_03_EU : Word := 1;
      pressure_04_EU : Word := 1;
      pressure_05_EU : Word := 1;
      pressure_06_EU : Word := 0;
      pressure_07_EU : Word := 0;
      pressure_08_EU : Word := 1;
      pressure_09_EU : Word := 1;
      pressure_10_EU : Word := 1;
      pressure_11_EU : Word := 3;
      pressure_12_EU : Word := 2;
      pressure_13_EU : Word := 0;
      pressure_14_EU : Word := 0;
      pressure_15_EU : Word := 3;
      pressure_16_EU : Word := 3;
      pressure_17_EU : Word := 3;
   END_VAR
BEGIN
END_DATA_BLOCK

DATA_BLOCK "PID_impulse_NAV_DB"   // DB245
{ S7_Optimized_Access := 'FALSE' }
VERSION : 0.1
// stored: InstanceOfName PID_impulse
"PID_impulse"
BEGIN
   DB := 0.5;
   KP := 0.18;
   TI := 4769;
   CYCLE := 100;
   FMT := 30000;
   DT_MIN := 127;
END_DATA_BLOCK

DATA_BLOCK "PID_impulse_NAD_DB"   // DB246
{ S7_Optimized_Access := 'FALSE' }
VERSION : 0.1
// stored: InstanceOfName PID_impulse
"PID_impulse"
BEGIN
   DB := 0.2;
   KP := 0.18;
   TI := 4891;
   CYCLE := 100;
   FMT := 33000;
   DT_MIN := 172;
END_DATA_BLOCK

DATA_BLOCK "PID_analog_DV_DB"   // DB256
{ S7_Optimized_Access := 'FALSE' }
VERSION : 0.1
// stored: InstanceOfName PID_analog
"PID_analog"
BEGIN
   DB := 10.0;
   KP := 0.05;
   TI := 10000;
   CYCLE := 100;
   OUT_MAX := 50.0;
END_DATA_BLOCK

DATA_BLOCK "PID_analog_DS_DB"   // DB258
{ S7_Optimized_Access := 'FALSE' }
VERSION : 0.1
// stored: InstanceOfName PID_analog
"PID_analog"
BEGIN
   DB := 2.0;
   KP := 0.05;
   TI := 3000;
   CYCLE := 100;
   OUT_MAX := 50.0;
END_DATA_BLOCK

DATA_BLOCK "PID_impulse_ZRW_DB"   // DB259
{ S7_Optimized_Access := 'FALSE' }
VERSION : 0.1
// stored: InstanceOfName PID_impulse
"PID_impulse"
BEGIN
END_DATA_BLOCK

DATA_BLOCK "Q_water"   // DB277
{ S7_Optimized_Access := 'FALSE' }
VERSION : 0.1
// Массовый расход воды (т/ч)
// stored: InstanceOfName Qm
"Qm"
BEGIN
   Enable := true;
   "a" := 0.6257558;
   Ksh := 1.00268;
   Kp := 1.01506;
   d := 24.719;
   ro := 943.9471;
END_DATA_BLOCK

DATA_BLOCK "Q_steam"   // DB282
{ S7_Optimized_Access := 'FALSE' }
VERSION : 0.1
// Массовый расход пара (т/ч)
// stored: InstanceOfName Qm_steam
"Qm_steam"
BEGIN
   Enable := true;
   d := 77.023;
   "a" := 0.6257204;
   Ksh := 1.00129;
   Kp := 1.00367;
   ro := 4.82808;
   Dtrub := 150.291;
   k := 1.141;
END_DATA_BLOCK

